(* IEC 61131-3 sources: study_plc/TimeStampFlat/content, 19 files *)

(* ---- main_prg.p~Variables~0000.var ---- *)
{ CustomGroupDefinition('a04e0da4-75a3-431c-a769-2ffcda83b779', '') }

VAR_EXTERNAL
    BUTTON_01 : BOOL { CustomGroupReference('a04e0da4-75a3-431c-a769-2ffcda83b779') } {Id('9d7c30a0-79f5-45dd-a2bb-9fe8afbc4b20')};
    LED : BOOL { CustomGroupReference('a04e0da4-75a3-431c-a769-2ffcda83b779') } {Id('db36f1cd-cd5f-4305-b62e-abae8295d826')};
END_VAR

VAR_GLOBAL
    bIsBlinking : BOOL { CustomGroupReference('a04e0da4-75a3-431c-a769-2ffcda83b779') } {Id('3276df67-48e3-40bd-b5cf-bc160ecd9fbf')};
    bLastButtonState : BOOL { CustomGroupReference('a04e0da4-75a3-431c-a769-2ffcda83b779') } {Id('10668f7e-212e-495e-babd-0d329f145ecd')};
    iBlinkCounter : INT { CustomGroupReference('a04e0da4-75a3-431c-a769-2ffcda83b779') } {Id('633e2c32-1f58-4700-8324-7b0311ee680d')};
    bCircleColor : BOOL { CustomGroupReference('a04e0da4-75a3-431c-a769-2ffcda83b779') } {Id('395212f8-a20c-46ba-a35b-0a9dcef59665')};
END_VAR

VAR_EXTERNAL
    counter : UINT { CustomGroupReference('a04e0da4-75a3-431c-a769-2ffcda83b779') } {Id('1701992e-3612-4291-8731-59990abaa8c7')};
    visual_counter : UINT { CustomGroupReference('a04e0da4-75a3-431c-a769-2ffcda83b779') } {Id('a891a596-3b4d-4571-8810-f9bcfd9d09ef')};
    tap_counter : UINT { CustomGroupReference('a04e0da4-75a3-431c-a769-2ffcda83b779') } {Id('a860a130-5121-4456-9e22-e20d3fb6a4d2')};
    TIMER : UINT { CustomGroupReference('a04e0da4-75a3-431c-a769-2ffcda83b779') } {Id('4b805dd1-1514-4363-b349-f760ae2ef950')};
    MESSAGE : BOOL { CustomGroupReference('a04e0da4-75a3-431c-a769-2ffcda83b779') } {Id('cdc6c82f-f8a2-467f-856e-2adb650c9a4f')};
    BUTTON_VIRTUAL : BOOL { CustomGroupReference('a04e0da4-75a3-431c-a769-2ffcda83b779') } {Id('e5aff69d-3d8e-4836-bed5-791e50e3ecc8')};
    buttonEdge : BOOL { CustomGroupReference('a04e0da4-75a3-431c-a769-2ffcda83b779') } {Id('871ce396-bc43-4252-ae3b-373c06ca63c2')};
    buttonCurrent : BOOL { CustomGroupReference('a04e0da4-75a3-431c-a769-2ffcda83b779') } {Id('1c2f3c40-a93c-4385-8462-9e9265ab8571')};
END_VAR

VAR
    FB21 : FB2 { CustomGroupReference('a04e0da4-75a3-431c-a769-2ffcda83b779') } {Id('54922560-dfac-4da8-a43d-80a38bc860ff')};
    FB22 : FB2 { CustomGroupReference('a04e0da4-75a3-431c-a769-2ffcda83b779') } {Id('0440c849-ac9a-4a62-b46c-6479d15f63f8')};
END_VAR

VAR_EXTERNAL
    TON_Blink : BOOL { CustomGroupReference('a04e0da4-75a3-431c-a769-2ffcda83b779') } {Id('319f1959-78a6-4cf2-81bc-d2dcea5df4e2')};
END_VAR

VAR
    FB23 : FB2 { CustomGroupReference('a04e0da4-75a3-431c-a769-2ffcda83b779') } {Id('546f7820-cb98-4ff5-a0ac-031b3fae9602')};
END_VAR

VAR_EXTERNAL
    blinkPeriod : UINT { CustomGroupReference('a04e0da4-75a3-431c-a769-2ffcda83b779') } {Id('be068b81-cd0d-40ca-b639-6780bc643a35')};
    TIME_TO_DINT : BOOL { CustomGroupReference('a04e0da4-75a3-431c-a769-2ffcda83b779') } {Id('cb415087-eb6f-4bb9-bdf8-b33e5cb765ee')};
    HMI_blinkPeriod : UINT { CustomGroupReference('a04e0da4-75a3-431c-a769-2ffcda83b779') } {Id('e62754f2-c4ad-4517-bcdd-83995e7e8a4c')};
END_VAR

VAR
    FB1 : FB { CustomGroupReference('a04e0da4-75a3-431c-a769-2ffcda83b779') } {Id('a21cc78b-fc91-401c-989f-5a3f00dbf2b6')};
    FB2 : FB { CustomGroupReference('a04e0da4-75a3-431c-a769-2ffcda83b779') } {Id('57562de0-dacc-42f6-93d3-63030d3f5b88')};
    FB3 : FB { CustomGroupReference('a04e0da4-75a3-431c-a769-2ffcda83b779') } {Id('74436edf-7137-4b89-ad20-294e1d8fb0ba')};
    FB4 : FB { CustomGroupReference('a04e0da4-75a3-431c-a769-2ffcda83b779') } {Id('58145396-09ad-45fc-99ee-1bc74df87d60')};
    FB5 : FB { CustomGroupReference('a04e0da4-75a3-431c-a769-2ffcda83b779') } {Id('605fd930-4c27-426e-82da-72f9c501b4c8')};
    UTC_in_Second1 : UTC_in_Second { CustomGroupReference('a04e0da4-75a3-431c-a769-2ffcda83b779') } {Id('561bc80b-119c-49be-b34c-1341fe2128dd')};
    UTC_in_Second2 : UTC_in_Second { CustomGroupReference('a04e0da4-75a3-431c-a769-2ffcda83b779') } {Id('187551ab-48a8-4595-8129-f3d7c5e3eedb')};
    UTC_in_Second3 : UTC_in_Second { CustomGroupReference('a04e0da4-75a3-431c-a769-2ffcda83b779') } {Id('8356627b-db3f-42a6-bade-665229c3f576')};
    UTC_in_Second4 : UTC_in_Second { CustomGroupReference('a04e0da4-75a3-431c-a769-2ffcda83b779') } {Id('4f025b1b-41c1-47cd-a402-58daae036f8e')};
    UTC_in_Second5 : UTC_in_Second { CustomGroupReference('a04e0da4-75a3-431c-a769-2ffcda83b779') } {Id('dae2764d-2f23-4bc9-8ce6-f3115f05c329')};
END_VAR

VAR_EXTERNAL
    TimestampMs : ULINT { CustomGroupReference('a04e0da4-75a3-431c-a769-2ffcda83b779') } {Id('bceea6ea-516d-42c0-a9bf-c36901277ad8')};
    ManualRTC : STRING { CustomGroupReference('a04e0da4-75a3-431c-a769-2ffcda83b779') } {Id('cec4a686-64db-40d8-a2d6-88bfda80289a')};
END_VAR

VAR
    UTC_in_Second6 : UTC_in_Second { CustomGroupReference('a04e0da4-75a3-431c-a769-2ffcda83b779') } {Id('34ce032f-88bf-46b0-9d48-2bfe1af360d8')};
END_VAR

(* ---- RES_3E844~GlobalVari~0000.var ---- *)
{ CustomGroupDefinition('fb84caa8-36a3-47d9-8bf0-95ff0e8a7b24', 'Default') }
{ CustomGroupDefinition('971398c9-e054-4349-a1d9-e00a1840c9f4', 'System Variables') }

VAR_GLOBAL
    BUTTON_01 : BOOL { CustomGroupReference('fb84caa8-36a3-47d9-8bf0-95ff0e8a7b24') } {Id('ff55c68f-4009-44e2-9111-0f6121b7f28e')};
    LED : BOOL { CustomGroupReference('fb84caa8-36a3-47d9-8bf0-95ff0e8a7b24') } {Id('a3518c0f-cfe9-4be8-920a-e2427bf7add7')};
    counter : UINT { CustomGroupReference('fb84caa8-36a3-47d9-8bf0-95ff0e8a7b24') } {Id('c758d767-5474-4789-9d22-781bfd7625a3')};
    bIsBlinking : BOOL { CustomGroupReference('fb84caa8-36a3-47d9-8bf0-95ff0e8a7b24') } {Id('41169e27-439a-46a2-bd00-94b8d785524f')};
    bLastButtonState : BOOL { CustomGroupReference('fb84caa8-36a3-47d9-8bf0-95ff0e8a7b24') } {Id('91fcfb61-3d5c-46c5-82ee-099172dd2d00')};
    visual_counter : UINT { CustomGroupReference('fb84caa8-36a3-47d9-8bf0-95ff0e8a7b24') } {Id('a5ecaf92-65ff-4985-a7f0-7e5144a773bc')};
    tap_counter : UINT { CustomGroupReference('fb84caa8-36a3-47d9-8bf0-95ff0e8a7b24') } {Id('7997c538-978c-452e-b505-3f3264cd3acb')};
    TIMER : UINT { CustomGroupReference('fb84caa8-36a3-47d9-8bf0-95ff0e8a7b24') } {Id('f51bd8e7-c0cd-421f-84a5-2d7e3e3f3667')};
    MESSAGE : BOOL { CustomGroupReference('fb84caa8-36a3-47d9-8bf0-95ff0e8a7b24') } {Id('3c2fc884-e19f-4beb-963f-04e6b1e4ad5f')};
    BUTTON_VIRTUAL : BOOL { CustomGroupReference('fb84caa8-36a3-47d9-8bf0-95ff0e8a7b24') } {Id('713492fe-22b0-4431-98a2-874f33c0214d')};
    buttonEdge : BOOL { CustomGroupReference('fb84caa8-36a3-47d9-8bf0-95ff0e8a7b24') } {Id('00cb1bf9-a75a-41ef-b864-ad11ab6e73bd')};
    buttonCurrent : BOOL { CustomGroupReference('fb84caa8-36a3-47d9-8bf0-95ff0e8a7b24') } {Id('a3914946-180c-4931-8b9b-c4945eb15232')};
END_VAR

VAR_CONFIG
    main_prg1.FB22.BUTTON_VIRTUAL : BOOL { InputLocation, CustomGroupReference('fb84caa8-36a3-47d9-8bf0-95ff0e8a7b24') } {Id('edaae17a-2832-4c67-ac45-b190593d386f')};
    main_prg1.FB21.BUTTON_VIRTUAL : BOOL { InputLocation, CustomGroupReference('fb84caa8-36a3-47d9-8bf0-95ff0e8a7b24') } {Id('30d0fe49-cb2f-4a7f-9de2-3afded5ed9e1')};
END_VAR

VAR_GLOBAL
    TIME_TO_DINT : BOOL { CustomGroupReference('fb84caa8-36a3-47d9-8bf0-95ff0e8a7b24') } {Id('c08fca2b-8685-447f-9b1d-964d4b9698af')};
    blinkPeriod : UINT { CustomGroupReference('fb84caa8-36a3-47d9-8bf0-95ff0e8a7b24') } {Id('a89eaa18-a4a3-4d70-906a-897dfc0313cd')};
    TON_Blink : BOOL { CustomGroupReference('fb84caa8-36a3-47d9-8bf0-95ff0e8a7b24') } {Id('687960f8-1ee0-416c-89ff-6b97b4efdd67')};
    HMI_blinkPeriod : UINT { CustomGroupReference('fb84caa8-36a3-47d9-8bf0-95ff0e8a7b24') } {Id('b5ffe9d3-7473-475f-903d-5c747d9fce23')};
    UINT_TO_TIME : BOOL { CustomGroupReference('fb84caa8-36a3-47d9-8bf0-95ff0e8a7b24') } {Id('56c9b7dd-8b0f-4834-bde7-82dd9a64a721')};
    PressStart : ULINT { CustomGroupReference('fb84caa8-36a3-47d9-8bf0-95ff0e8a7b24') } {Id('72598318-5edc-48d2-b4c1-9021699f7749')};
    PressTime : ULINT { CustomGroupReference('fb84caa8-36a3-47d9-8bf0-95ff0e8a7b24') } {Id('20e9929e-5bd7-41be-87ae-dc1696108355')};
    bButton : BOOL { CustomGroupReference('fb84caa8-36a3-47d9-8bf0-95ff0e8a7b24') } {Id('1b65edaf-19e7-4e96-9bb3-230a0c218b20')};
    BlinkReset : BOOL { CustomGroupReference('fb84caa8-36a3-47d9-8bf0-95ff0e8a7b24') } {Id('49695894-1423-4474-9eaa-ce1ad988c3f5')};
    test_us_1 : ULINT { CustomGroupReference('fb84caa8-36a3-47d9-8bf0-95ff0e8a7b24') } {Id('b3f01b14-7269-48aa-a0bd-12850281ca48')};
    test_us_2 : ULINT { CustomGroupReference('fb84caa8-36a3-47d9-8bf0-95ff0e8a7b24') } {Id('3fb0d77d-6462-4922-9943-9df0e6459224')};
    sTime : STRING { CustomGroupReference('fb84caa8-36a3-47d9-8bf0-95ff0e8a7b24') } {Id('b1cc24f8-6954-4e78-a01b-3fb7d85319ce')};
    bRTC_Ready : BOOL { CustomGroupReference('fb84caa8-36a3-47d9-8bf0-95ff0e8a7b24') } {Id('517801c9-9df0-49bf-9626-1117f62db573')};
    nLastBlink : ULINT { CustomGroupReference('fb84caa8-36a3-47d9-8bf0-95ff0e8a7b24') } {Id('f0fc7b48-9d55-4261-81d7-a2b4516753ed')};
    debug_toggle : INT { CustomGroupReference('fb84caa8-36a3-47d9-8bf0-95ff0e8a7b24') } {Id('4f1d6557-6d1f-4585-8eaa-0d52a0a13aa6')};
    bVirtualPulse : BOOL { CustomGroupReference('fb84caa8-36a3-47d9-8bf0-95ff0e8a7b24') } {Id('1a3d1420-8400-4ed1-ae9a-b1be359f92a0')};
    bLastVirtual : BOOL { CustomGroupReference('fb84caa8-36a3-47d9-8bf0-95ff0e8a7b24') } {Id('2a59c38b-860d-41cc-b434-8815cd6eb838')};
    bVirtTrig : BOOL { CustomGroupReference('fb84caa8-36a3-47d9-8bf0-95ff0e8a7b24') } {Id('2d522a4e-02e2-4d08-8e87-e2abe91557be')};
    bLastButton : BOOL { CustomGroupReference('fb84caa8-36a3-47d9-8bf0-95ff0e8a7b24') } {Id('e926f615-f63b-44f9-a00b-60eff743de3b')};
    rTrigVirt : BOOL { CustomGroupReference('fb84caa8-36a3-47d9-8bf0-95ff0e8a7b24') } {Id('95be6528-0073-416e-87ec-9c3c74cfbb9f')};
    rTrigPhys : BOOL { CustomGroupReference('fb84caa8-36a3-47d9-8bf0-95ff0e8a7b24') } {Id('f3b9ac2f-ae6f-4cfb-9b98-34b4fd9e6e43')};
    bWaitForRelease : BOOL { CustomGroupReference('fb84caa8-36a3-47d9-8bf0-95ff0e8a7b24') } {Id('cee13b13-a0ba-47f2-85b5-a1153d2bfc4d')};
    bLastPhys : BOOL { CustomGroupReference('fb84caa8-36a3-47d9-8bf0-95ff0e8a7b24') } {Id('2c93ea6f-76fc-46c1-8245-239521de7509')};
    bLastVirt : BOOL { CustomGroupReference('fb84caa8-36a3-47d9-8bf0-95ff0e8a7b24') } {Id('e15edbd4-dc20-4abf-a76b-535e03ed0216')};
    bVirtOneShot : BOOL { CustomGroupReference('fb84caa8-36a3-47d9-8bf0-95ff0e8a7b24') } {Id('180e95ba-7660-42f3-ab82-8aa1f4af8f65')};
    bPhysOneShot : BOOL { CustomGroupReference('fb84caa8-36a3-47d9-8bf0-95ff0e8a7b24') } {Id('b17a499a-a16a-4e07-a451-effc40a9126b')};
    bAnyPress : BOOL { CustomGroupReference('fb84caa8-36a3-47d9-8bf0-95ff0e8a7b24') } {Id('0312dcf0-9424-407f-a37e-e022e10eb398')};
    bVirtOld : BOOL { CustomGroupReference('fb84caa8-36a3-47d9-8bf0-95ff0e8a7b24') } {Id('ca6bffc0-4800-4d66-aefe-acab4512e9e1')};
    TRIM : BOOL { CustomGroupReference('fb84caa8-36a3-47d9-8bf0-95ff0e8a7b24') } {Id('6c8b045d-0aab-487b-b1ad-cb855cf61a63')};
    bRTCReady : BOOL { CustomGroupReference('fb84caa8-36a3-47d9-8bf0-95ff0e8a7b24') } {Id('cb59c76f-3031-4077-8f90-714e8f7a8c8b')};
    TimestampMs : ULINT { CustomGroupReference('fb84caa8-36a3-47d9-8bf0-95ff0e8a7b24') } {Id('84cfde2f-c5c3-4348-808e-c1645fed4d81')};
    TimeZone : INT { CustomGroupReference('fb84caa8-36a3-47d9-8bf0-95ff0e8a7b24') } {Id('1288d1f3-3ab3-4651-8a72-0030e0acb8f2')};
    nTimeZoneOffset : INT { CustomGroupReference('fb84caa8-36a3-47d9-8bf0-95ff0e8a7b24') } {Id('d52ba4d7-7e69-49ff-be6d-e2df38c82290')};
    sOutputDate : STRING { CustomGroupReference('fb84caa8-36a3-47d9-8bf0-95ff0e8a7b24') } {Id('045fa39e-965c-40ad-9d1c-b2ae0bfc88d7')};
    ulInputMS : ULINT { CustomGroupReference('fb84caa8-36a3-47d9-8bf0-95ff0e8a7b24') } {Id('57f31c1f-ce8e-4e9a-a54f-91a1926557d9')};
    sCustomDate : STRING { CustomGroupReference('fb84caa8-36a3-47d9-8bf0-95ff0e8a7b24') } {Id('7e064ee7-e4f6-4547-b34e-d6702123f182')};
END_VAR

VAR_CONFIG
    main_prg1.UTC_in_Second5.DaysInMonth : INT { InputLocation, CustomGroupReference('fb84caa8-36a3-47d9-8bf0-95ff0e8a7b24') } {Id('0b54d02d-88a7-4f64-a714-37ba5a4d2863')};
    main_prg1.UTC_in_Second4.DaysInMonth : INT { InputLocation, CustomGroupReference('fb84caa8-36a3-47d9-8bf0-95ff0e8a7b24') } {Id('c5c31dc5-7259-4959-b722-8cf1dc1f7ee6')};
    main_prg1.UTC_in_Second3.DaysInMonth : INT { InputLocation, CustomGroupReference('fb84caa8-36a3-47d9-8bf0-95ff0e8a7b24') } {Id('babf101c-e82f-4d04-9ab9-a52ee78929ee')};
    main_prg1.UTC_in_Second2.DaysInMonth : INT { InputLocation, CustomGroupReference('fb84caa8-36a3-47d9-8bf0-95ff0e8a7b24') } {Id('af5cefd6-4978-424f-95ca-eec832feb9ce')};
    main_prg1.UTC_in_Second1.DaysInMonth : INT { InputLocation, CustomGroupReference('fb84caa8-36a3-47d9-8bf0-95ff0e8a7b24') } {Id('cc2d7a49-7d34-4f98-8bad-cdc305743582')};
END_VAR

VAR_GLOBAL
    sTmp : BOOL { CustomGroupReference('fb84caa8-36a3-47d9-8bf0-95ff0e8a7b24') } {Id('52421147-2409-4498-864b-2a037dc35c02')};
    sTmp2 : BOOL { CustomGroupReference('fb84caa8-36a3-47d9-8bf0-95ff0e8a7b24') } {Id('9060f604-83ec-4e2e-8322-d678c276741c')};
    sYy : STRING { CustomGroupReference('fb84caa8-36a3-47d9-8bf0-95ff0e8a7b24') } {Id('4c9b6b92-2451-4146-be8f-061a9e49ac85')};
    sMo : STRING { CustomGroupReference('fb84caa8-36a3-47d9-8bf0-95ff0e8a7b24') } {Id('2338197b-f5fd-40a7-9e1a-48057039073d')};
    nMonthDays : INT { CustomGroupReference('fb84caa8-36a3-47d9-8bf0-95ff0e8a7b24') } {Id('afdd7226-203a-4163-8ab4-f50e96edd491')};
    UseManualRTC : BOOL { CustomGroupReference('fb84caa8-36a3-47d9-8bf0-95ff0e8a7b24') } {Id('b1822fe9-4cea-4d3a-b67e-cfc11819dcf7')};
    ManualRTC : STRING { CustomGroupReference('fb84caa8-36a3-47d9-8bf0-95ff0e8a7b24') } {Id('03a235b0-b550-43e6-9f6e-0f7724ebddc2')};
    TimezoneOffset : INT { CustomGroupReference('fb84caa8-36a3-47d9-8bf0-95ff0e8a7b24') } {Id('24b06e47-b007-45e8-8735-7f3f73c4efa8')};
END_VAR

VAR_CONFIG
    main_prg1.UTC_in_Second6.DaysInMonth : INT { InputLocation, CustomGroupReference('fb84caa8-36a3-47d9-8bf0-95ff0e8a7b24') } {Id('18a8efd7-5980-422a-b2ec-fcc23db0160e')};
END_VAR

VAR_GLOBAL
    PND_S1_PLC_RUN : BOOL { SystemVariable, CustomGroupReference('971398c9-e054-4349-a1d9-e00a1840c9f4') } {Id('a8109aaa-718e-4ad7-9ef6-414f49af5f2c')}; (*Higher level PLC in RUN*)
    PND_S1_VALID_DATA_CYCLE : BOOL { SystemVariable, CustomGroupReference('971398c9-e054-4349-a1d9-e00a1840c9f4') } {Id('e4636e3b-85f5-4518-8ba6-e632d844bd79')}; (*Connection to Profinet-Controller*)
    PND_S1_OUTPUT_STATUS_GOOD : BOOL { SystemVariable, CustomGroupReference('971398c9-e054-4349-a1d9-e00a1840c9f4') } {Id('9e967e71-8e8f-40d9-aae6-a7f87e15c1dc')}; (*IOP status of the higher-level control system*)
    PND_S1_INPUT_STATUS_GOOD : BOOL { SystemVariable, CustomGroupReference('971398c9-e054-4349-a1d9-e00a1840c9f4') } {Id('b1e203c1-a3c2-41a1-8f15-cba8c60dc0f2')}; (*IOC status of the higher-level control system*)
    PND_S1_DATA_LENGTH : WORD { SystemVariable, CustomGroupReference('971398c9-e054-4349-a1d9-e00a1840c9f4') } {Id('c69796fa-e3a1-44c3-8dc7-85a985bef384')}; (*Process data length*)
    PND_S1_OUTPUTS : PND_IO_512 { SystemVariable, CustomGroupReference('971398c9-e054-4349-a1d9-e00a1840c9f4'), Assignable(IsWritable := True), Origin('epd056') } {Id('871d0d2f-9f74-43af-844e-7e8a0b6267c3')}; (*Output process data*)
    PND_S1_INPUTS : PND_IO_512 { SystemVariable, CustomGroupReference('971398c9-e054-4349-a1d9-e00a1840c9f4') } {Id('26de38c2-6476-4746-acc5-bee0b9f2dbfa')}; (*Input process data*)
    PND_IO_DRIVEN_BY_PLC : INT { SystemVariable, CustomGroupReference('971398c9-e054-4349-a1d9-e00a1840c9f4') } {Id('00739d06-8933-4fec-8048-b3cebcbc2058')};
    AXIO_DIAG_STATUS_REG_HI : BYTE { SystemVariable, CustomGroupReference('971398c9-e054-4349-a1d9-e00a1840c9f4') } {Id('4f9c59a1-643a-4475-a439-ad1cf8561ad6')};
    AXIO_DIAG_STATUS_REG_LOW : BYTE { SystemVariable, CustomGroupReference('971398c9-e054-4349-a1d9-e00a1840c9f4') } {Id('eae2279f-0f04-4890-a0bf-b55fad2d0afa')};
    AXIO_DIAG_PARAM_REG_HI : BYTE { SystemVariable, CustomGroupReference('971398c9-e054-4349-a1d9-e00a1840c9f4') } {Id('0caba1d5-e173-4e1b-b805-00d054efa100')};
    AXIO_DIAG_PARAM_REG_LOW : BYTE { SystemVariable, CustomGroupReference('971398c9-e054-4349-a1d9-e00a1840c9f4') } {Id('67315ed2-b4f9-44bb-859d-233dd4b3c9bb')};
    AXIO_DIAG_PARAM_2_REG_HI : BYTE { SystemVariable, CustomGroupReference('971398c9-e054-4349-a1d9-e00a1840c9f4') } {Id('981f8143-c142-4f6c-ae92-2b18592edb2f')};
    AXIO_DIAG_PARAM_2_REG_LOW : BYTE { SystemVariable, CustomGroupReference('971398c9-e054-4349-a1d9-e00a1840c9f4') } {Id('f7a3077a-9e70-458b-acdb-2714bd9d86a3')};
    AXIO_DIAG_STATUS_REG_PF : BOOL { SystemVariable, CustomGroupReference('971398c9-e054-4349-a1d9-e00a1840c9f4') } {Id('c49d1a45-1fcc-4ae2-b55e-619e93c6f775')};
    AXIO_DIAG_STATUS_REG_BUS : BOOL { SystemVariable, CustomGroupReference('971398c9-e054-4349-a1d9-e00a1840c9f4') } {Id('17b3305e-f37e-4a9d-94a4-5a3d9ca6ad1a')};
    AXIO_DIAG_STATUS_REG_RUN : BOOL { SystemVariable, CustomGroupReference('971398c9-e054-4349-a1d9-e00a1840c9f4') } {Id('79b3d4f7-46d4-4c7b-aa70-24e501b5afeb')};
    AXIO_DIAG_STATUS_REG_ACT : BOOL { SystemVariable, CustomGroupReference('971398c9-e054-4349-a1d9-e00a1840c9f4') } {Id('a0315e8d-4040-4508-b50d-7fa5ad74f7a1')};
    AXIO_DIAG_STATUS_REG_RDY : BOOL { SystemVariable, CustomGroupReference('971398c9-e054-4349-a1d9-e00a1840c9f4') } {Id('c8b37275-37bf-40c1-94c8-2d91ca269131')};
    AXIO_DIAG_STATUS_REG_SYSFAIL : BOOL { SystemVariable, CustomGroupReference('971398c9-e054-4349-a1d9-e00a1840c9f4') } {Id('a230509c-5098-49c0-94c0-ee773a64e2de')};
    AXIO_DIAG_STATUS_REG_PW : BOOL { SystemVariable, CustomGroupReference('971398c9-e054-4349-a1d9-e00a1840c9f4') } {Id('67e3682d-83f4-44e0-ac88-2f95bae65960')};
    IB_DIAG_STATUS_REG_HI : BYTE { SystemVariable, CustomGroupReference('971398c9-e054-4349-a1d9-e00a1840c9f4'), Assignable(IsWritable := True), Origin('epdib1') } {Id('870f34b1-cbfb-4a12-9a3a-674532964b8e')};
    IB_DIAG_STATUS_REG_LOW : BYTE { SystemVariable, CustomGroupReference('971398c9-e054-4349-a1d9-e00a1840c9f4'), Assignable(IsWritable := True), Origin('epdib2') } {Id('6aca7f7b-4495-47d2-b6c9-b992b56c11ef')};
    IB_DIAG_STATUS_REG_SYSFAIL : BOOL { SystemVariable, CustomGroupReference('971398c9-e054-4349-a1d9-e00a1840c9f4'), Assignable(IsWritable := True), Origin('epdib3') } {Id('8836a82b-e65b-4bcd-bdda-0e80ed208fef')};
    IB_DIAG_STATUS_REG_WARN : BOOL { SystemVariable, CustomGroupReference('971398c9-e054-4349-a1d9-e00a1840c9f4'), Assignable(IsWritable := True), Origin('epdib4') } {Id('590ff5fc-a4de-4153-abff-4c319033e938')};
    IB_DIAG_STATUS_REG_QUAL : BOOL { SystemVariable, CustomGroupReference('971398c9-e054-4349-a1d9-e00a1840c9f4'), Assignable(IsWritable := True), Origin('epdib5') } {Id('016a54f4-214c-4108-9e23-713c4e30776f')};
    IB_DIAG_STATUS_REG_USER : BOOL { SystemVariable, CustomGroupReference('971398c9-e054-4349-a1d9-e00a1840c9f4'), Assignable(IsWritable := True), Origin('epdib6') } {Id('436892d9-24f4-4bde-b365-39ce805afbcb')};
    IB_DIAG_STATUS_REG_PF : BOOL { SystemVariable, CustomGroupReference('971398c9-e054-4349-a1d9-e00a1840c9f4'), Assignable(IsWritable := True), Origin('epdib7') } {Id('9db6ace2-a1c0-4f18-b2cc-23c676225b79')};
    IB_DIAG_STATUS_REG_BUS : BOOL { SystemVariable, CustomGroupReference('971398c9-e054-4349-a1d9-e00a1840c9f4'), Assignable(IsWritable := True), Origin('epdib8') } {Id('69b61899-e7d4-45a0-a00c-0858c7e6436a')};
    IB_DIAG_STATUS_REG_CTRL : BOOL { SystemVariable, CustomGroupReference('971398c9-e054-4349-a1d9-e00a1840c9f4'), Assignable(IsWritable := True), Origin('epdib9') } {Id('ea44b33b-9512-4145-9c83-f5fc837d58a5')};
    IB_DIAG_STATUS_REG_DTC : BOOL { SystemVariable, CustomGroupReference('971398c9-e054-4349-a1d9-e00a1840c9f4'), Assignable(IsWritable := True), Origin('epdib10') } {Id('56dd80ec-9280-441e-bd4f-2ac40a37e096')};
    IB_DIAG_STATUS_REG_RUN : BOOL { SystemVariable, CustomGroupReference('971398c9-e054-4349-a1d9-e00a1840c9f4'), Assignable(IsWritable := True), Origin('epdib11') } {Id('c59a357f-adc9-49ca-a807-b1c10b0d67a2')};
    IB_DIAG_STATUS_REG_ACT : BOOL { SystemVariable, CustomGroupReference('971398c9-e054-4349-a1d9-e00a1840c9f4'), Assignable(IsWritable := True), Origin('epdib12') } {Id('e3ecf724-72f2-4fe3-be90-c451638ac496')};
    IB_DIAG_STATUS_REG_RDY : BOOL { SystemVariable, CustomGroupReference('971398c9-e054-4349-a1d9-e00a1840c9f4'), Assignable(IsWritable := True), Origin('epdib13') } {Id('5c061d11-60fc-4a47-a192-85e8775eb15f')};
    IB_DIAG_PARAM_REG_HI : BYTE { SystemVariable, CustomGroupReference('971398c9-e054-4349-a1d9-e00a1840c9f4'), Assignable(IsWritable := True), Origin('epdib14') } {Id('38a23e35-1cd8-4d9c-96d6-810c618d5526')};
    IB_DIAG_PARAM_REG_LOW : BYTE { SystemVariable, CustomGroupReference('971398c9-e054-4349-a1d9-e00a1840c9f4'), Assignable(IsWritable := True), Origin('epdib15') } {Id('5b495f5b-d26e-4cff-836b-0fe238b1654d')};
    IB_DIAG_PARAM_2_REG_HI : BYTE { SystemVariable, CustomGroupReference('971398c9-e054-4349-a1d9-e00a1840c9f4'), Assignable(IsWritable := True), Origin('epdib16') } {Id('317a6edf-8d30-4505-8601-eb0d20c3c6e2')};
    IB_DIAG_PARAM_2_REG_LOW : BYTE { SystemVariable, CustomGroupReference('971398c9-e054-4349-a1d9-e00a1840c9f4'), Assignable(IsWritable := True), Origin('epdib17') } {Id('83c1a718-f3e7-4cc0-841f-c1e2233f8d2e')};
    ESM_DATA : ESM_DAT { SystemVariable, CustomGroupReference('971398c9-e054-4349-a1d9-e00a1840c9f4'), Assignable(IsWritable := True), Origin('epd100') } {Id('74de6c32-cd1d-4959-95c5-ec365806a030')};
    RTC : RTC_TYPE { SystemVariable, CustomGroupReference('971398c9-e054-4349-a1d9-e00a1840c9f4') } {Id('3c52e428-0cdb-4c6c-bc54-e6da1e8c50fe')};
    DEVICE_STATE : DEVICE_STATE_2152_TYPE { SystemVariable, CustomGroupReference('971398c9-e054-4349-a1d9-e00a1840c9f4') } {Id('1129891b-b5a9-4d3b-b9a0-4936e33ad606')};
    USER_PARTITION : PARTITION_INFO { SystemVariable, CustomGroupReference('971398c9-e054-4349-a1d9-e00a1840c9f4') } {Id('4b7f6b3b-3696-419a-a21a-ce7cb6ceb9db')};
    PNIO_SYSTEM_BF : BOOL { SystemVariable, CustomGroupReference('971398c9-e054-4349-a1d9-e00a1840c9f4') } {Id('ea9f164c-d192-4b60-b66f-cf87b53d5e5b')};
    PNIO_SYSTEM_SF : BOOL { SystemVariable, CustomGroupReference('971398c9-e054-4349-a1d9-e00a1840c9f4') } {Id('de2bebd9-d808-496f-954f-38ec8ace12e8')};
    PNIO_MAINTENANCE_DEMANDED : BOOL { SystemVariable, CustomGroupReference('971398c9-e054-4349-a1d9-e00a1840c9f4') } {Id('4c4c4e79-3946-4f32-b468-22905a5c8f5f')};
    PNIO_MAINTENANCE_REQUIRED : BOOL { SystemVariable, CustomGroupReference('971398c9-e054-4349-a1d9-e00a1840c9f4') } {Id('0dfc99eb-ecfe-45c6-afb8-64b2d7705677')};
    PNIO_CONFIG_STATUS : WORD { SystemVariable, CustomGroupReference('971398c9-e054-4349-a1d9-e00a1840c9f4') } {Id('c34f805f-b5c2-44af-bb0f-7c49d4666c2f')};
    PNIO_CONFIG_STATUS_ACTIVE : BOOL { SystemVariable, CustomGroupReference('971398c9-e054-4349-a1d9-e00a1840c9f4') } {Id('d08caa2c-5061-4764-8b36-3a6b79934353')};
    PNIO_CONFIG_STATUS_READY : BOOL { SystemVariable, CustomGroupReference('971398c9-e054-4349-a1d9-e00a1840c9f4') } {Id('25aaf986-14d2-455e-8fb6-e8e35bd65063')};
    PNIO_CONFIG_STATUS_CFG_FAULT : BOOL { SystemVariable, CustomGroupReference('971398c9-e054-4349-a1d9-e00a1840c9f4') } {Id('7223f36b-f452-48c9-a964-10165bc7f0a7')};
    PNIO_FORCE_FAILSAFE : BOOL { SystemVariable, CustomGroupReference('971398c9-e054-4349-a1d9-e00a1840c9f4'), Assignable(IsWritable := True), Origin('epd145') } {Id('e1337b3e-a988-48a5-87ec-e8461474d15f')};
    PNIO_FORCE_PRIMARY : BOOL { SystemVariable, CustomGroupReference('971398c9-e054-4349-a1d9-e00a1840c9f4'), Assignable(IsWritable := True), Origin('epd159') } {Id('2e5ecda8-89ea-46e5-93c1-a46de4cc3fa2')};
    IP_ACTIVE_SOCKETS AT %MW1.30000 : UINT { SystemVariable, CustomGroupReference('971398c9-e054-4349-a1d9-e00a1840c9f4') } {Id('f10f644a-6de6-4578-8707-c22090109bfe')};
    TLS_ACTIVE_SOCKETS AT %MW1.30100 : UINT { SystemVariable, CustomGroupReference('971398c9-e054-4349-a1d9-e00a1840c9f4') } {Id('b614145a-4322-4555-8406-73f21140d7b8')};
    HMI_STATUS2 : HMI_STATUS_TYPE2 { SystemVariable, CustomGroupReference('971398c9-e054-4349-a1d9-e00a1840c9f4') } {Id('a142712d-5d2f-43da-8c93-deb2c52e6525')};
    HMI_CONTROL : HMI_CONTROL_TYPE { SystemVariable, CustomGroupReference('971398c9-e054-4349-a1d9-e00a1840c9f4'), Assignable(IsWritable := True), Origin('epd151') } {Id('9e0c5809-738c-47e0-98c3-088c020b755a')};
    EIPD_INPUTS : EIPD_IO_ARRAY { SystemVariable, CustomGroupReference('971398c9-e054-4349-a1d9-e00a1840c9f4') } {Id('876bd6bd-0ab9-42a0-8c1a-986f5c03e455')};
    EIPD_OUTPUTS : EIPD_IO_ARRAY { SystemVariable, CustomGroupReference('971398c9-e054-4349-a1d9-e00a1840c9f4'), Assignable(IsWritable := True), Origin('epd153') } {Id('ee7a2a99-783e-472f-9cae-c449c38f3da8')};
    EIPD_VALID_DATA_CYCLE : BOOL { SystemVariable, CustomGroupReference('971398c9-e054-4349-a1d9-e00a1840c9f4') } {Id('7ef7e2c3-a29c-4fb9-b6b9-6d2708115b6c')};
    EIPD_PEER_IDLE : BOOL { SystemVariable, CustomGroupReference('971398c9-e054-4349-a1d9-e00a1840c9f4') } {Id('ece7b39f-4744-4856-ab49-ac0106b18a4c')};
    EIPD_PEER_RUN : BOOL { SystemVariable, CustomGroupReference('971398c9-e054-4349-a1d9-e00a1840c9f4') } {Id('9a9a04d6-b3b6-4f81-8713-309c56ef942d')};
    EIPD_OUTPUTS_LENGTH : WORD { SystemVariable, CustomGroupReference('971398c9-e054-4349-a1d9-e00a1840c9f4') } {Id('852a06b4-24e7-4a6a-a226-9832b61a169c')};
    EIPD_INPUTS_LENGTH : WORD { SystemVariable, CustomGroupReference('971398c9-e054-4349-a1d9-e00a1840c9f4') } {Id('2475dd19-5aff-47a6-ba79-1133d75b5c3e')};
    PLC_CRC_PRJ AT %ML1.10000 : ULINT { SystemVariable, CustomGroupReference('971398c9-e054-4349-a1d9-e00a1840c9f4') } {Id('41b139bc-2750-4dde-b5bf-ab57e61bf63e')};
END_VAR

(* ---- FB.pou~Code~0000.st ---- *)
// время с контроллера
fbRTC(EN := TRUE, CDT => sTime, Q => bRTC_Ready);

// парс
fbParseTime(
    sTime := sTime,
    Year => nYear,
    Month => nMonth,
    Day => nDay,
    Hour => nHour,
    Minute => nMinute,
    Second => nSecond,
    Millisecond => nMS,
    Valid => bTimeValid
);

// количество дней от 1970
nDays := 0;

FOR i := 1970 TO nYear - 1 DO
    IF ((i MOD 4 = 0) AND (i MOD 100 <> 0)) OR (i MOD 400 = 0) THEN
        nDays := nDays + 366;
    ELSE
        nDays := nDays + 365;
    END_IF;
END_FOR;

// добавляем дни за полные месяцы
IF nMonth > 1 THEN nDays := nDays + 31; END_IF;
IF nMonth > 2 THEN
    IF ((nYear MOD 4 = 0) AND (nYear MOD 100 <> 0)) OR (nYear MOD 400 = 0) THEN
        nDays := nDays + 29;
    ELSE
        nDays := nDays + 28;
    END_IF;
END_IF;
IF nMonth > 3 THEN nDays := nDays + 31; END_IF;
IF nMonth > 4 THEN nDays := nDays + 30; END_IF;
IF nMonth > 5 THEN nDays := nDays + 31; END_IF;
IF nMonth > 6 THEN nDays := nDays + 30; END_IF;
IF nMonth > 7 THEN nDays := nDays + 31; END_IF;
IF nMonth > 8 THEN nDays := nDays + 31; END_IF;
IF nMonth > 9 THEN nDays := nDays + 30; END_IF;
IF nMonth > 10 THEN nDays := nDays + 31; END_IF;
IF nMonth > 11 THEN nDays := nDays + 30; END_IF;

// добавим дни текущего месяца
nDays := nDays + (nDay - 1);

// перевод всё в мс
TimestampMs :=
    DINT_TO_ULINT(nDays) * 86400000 +
    INT_TO_ULINT(nHour) * 3600000 +
    INT_TO_ULINT(nMinute) * 60000 +
    INT_TO_ULINT(nSecond) * 1000 +
    INT_TO_ULINT(nMS);

// сброс
IF BlinkReset THEN
    bIsBlinking := FALSE;
    visual_counter := 0;
    tap_counter := 0;
    LED := FALSE;
    nLastBlink := 0;
    bWaitForRelease := FALSE;
    BlinkReset := FALSE;
END_IF

(* ---- FB.pou~Variables~0000.var ---- *)
{ CustomGroupDefinition('d879d638-e7f1-4a28-a2ab-b4cf2ec7bb4a', '') }

VAR_INPUT
    BUTTON_01 : BOOL { CustomGroupReference('d879d638-e7f1-4a28-a2ab-b4cf2ec7bb4a') } {Id('4e0719f1-9a21-49b0-ab1a-7bca753de8bf')};
    BUTTON_VIRTUAL : BOOL { CustomGroupReference('d879d638-e7f1-4a28-a2ab-b4cf2ec7bb4a') } {Id('16b13fcd-91ca-4fbd-bce8-5329faf97148')};
END_VAR

VAR_OUTPUT
    LED : BOOL { CustomGroupReference('d879d638-e7f1-4a28-a2ab-b4cf2ec7bb4a') } {Id('35a522c3-a831-4de5-82d7-ae5b3c0dd537')};
    MESSAGE : BOOL { CustomGroupReference('d879d638-e7f1-4a28-a2ab-b4cf2ec7bb4a') } {Id('fb214dee-66f6-463f-9713-862a6108447e')};
END_VAR

VAR
    PressStart : ULINT { CustomGroupReference('d879d638-e7f1-4a28-a2ab-b4cf2ec7bb4a') } {Id('ae5033d3-fed2-43d0-adf6-ccfa772e577f')};
    PressTime : ULINT { CustomGroupReference('d879d638-e7f1-4a28-a2ab-b4cf2ec7bb4a') } {Id('67c05195-0624-4f5b-a4a4-63254ac533c9')};
    bButton : BOOL { CustomGroupReference('d879d638-e7f1-4a28-a2ab-b4cf2ec7bb4a') } {Id('a6f25af8-da50-4153-a6f2-77781ed29851')};
    bLastButtonState : BOOL { CustomGroupReference('d879d638-e7f1-4a28-a2ab-b4cf2ec7bb4a') } {Id('4f0463dc-8f77-4d98-87a2-aa94574099e2')};
    bIsBlinking : BOOL { CustomGroupReference('d879d638-e7f1-4a28-a2ab-b4cf2ec7bb4a') } {Id('b9bf86c3-b159-4991-9861-6f5314b0321c')};
    BlinkReset : BOOL { CustomGroupReference('d879d638-e7f1-4a28-a2ab-b4cf2ec7bb4a') } {Id('7e2c85d6-cf72-46e0-b9a5-424ab27580a5')};
    TON_Blink : TON { CustomGroupReference('d879d638-e7f1-4a28-a2ab-b4cf2ec7bb4a') } {Id('197c8782-f631-4ffa-a13c-2cd90675b891')};
END_VAR

VAR_EXTERNAL
    visual_counter : UINT { CustomGroupReference('d879d638-e7f1-4a28-a2ab-b4cf2ec7bb4a') } {Id('ed5c4f7a-75fb-4186-8b26-909a554518ed')};
    tap_counter : UINT { CustomGroupReference('d879d638-e7f1-4a28-a2ab-b4cf2ec7bb4a') } {Id('8e4fb33c-aed4-48aa-8ee2-6ffca498c8a3')};
END_VAR

VAR
    dummy : ULINT { CustomGroupReference('d879d638-e7f1-4a28-a2ab-b4cf2ec7bb4a') } {Id('206ff9a5-ceb4-427d-bf17-5ced64b3d33f')};
    fbRTC : RTC_S { CustomGroupReference('d879d638-e7f1-4a28-a2ab-b4cf2ec7bb4a') } {Id('689cfebd-229e-4b45-8dd0-65fa994717f3')};
END_VAR

VAR_EXTERNAL
    sTime : STRING { CustomGroupReference('d879d638-e7f1-4a28-a2ab-b4cf2ec7bb4a') } {Id('91bb18d7-44e6-4613-a079-9ddb7a779d7d')};
    bRTC_Ready : BOOL { CustomGroupReference('d879d638-e7f1-4a28-a2ab-b4cf2ec7bb4a') } {Id('c414b8d8-2513-4024-ae96-ac7c04fab89d')};
    nLastBlink : ULINT { CustomGroupReference('d879d638-e7f1-4a28-a2ab-b4cf2ec7bb4a') } {Id('cb3e5d71-9c5a-4d71-8037-b20658097fc0')};
    debug_toggle : INT { CustomGroupReference('d879d638-e7f1-4a28-a2ab-b4cf2ec7bb4a') } {Id('2072d667-54cb-490a-b42a-0cae67e0ad60')};
    bVirtualPulse : BOOL { CustomGroupReference('d879d638-e7f1-4a28-a2ab-b4cf2ec7bb4a') } {Id('6798c4c2-251a-4f23-8819-dd3632552722')};
    bLastVirtual : BOOL { CustomGroupReference('d879d638-e7f1-4a28-a2ab-b4cf2ec7bb4a') } {Id('53ac58ec-322e-422e-aaf0-86794f043220')};
    bVirtTrig : BOOL { CustomGroupReference('d879d638-e7f1-4a28-a2ab-b4cf2ec7bb4a') } {Id('57ff68d4-c262-4da7-a951-55c5bc88e074')};
    bLastButton : BOOL { CustomGroupReference('d879d638-e7f1-4a28-a2ab-b4cf2ec7bb4a') } {Id('3a263dd4-d980-4a3f-9643-d60d3c28d595')};
END_VAR

VAR
    rTrigVirt : R_TRIG { CustomGroupReference('d879d638-e7f1-4a28-a2ab-b4cf2ec7bb4a') } {Id('c425a54f-4ffb-481e-90de-1a6ced1796a6')};
    rTrigPhys : R_TRIG { CustomGroupReference('d879d638-e7f1-4a28-a2ab-b4cf2ec7bb4a') } {Id('19454729-86e8-4c30-9d95-3b307f57250b')};
END_VAR

VAR_EXTERNAL
    bWaitForRelease : BOOL { CustomGroupReference('d879d638-e7f1-4a28-a2ab-b4cf2ec7bb4a') } {Id('f76a665a-d697-43fa-a6b8-18f2ea8978be')};
    bLastPhys : BOOL { CustomGroupReference('d879d638-e7f1-4a28-a2ab-b4cf2ec7bb4a') } {Id('531aa2b4-5bc9-4d3d-a0a4-8ab213c87f93')};
    bLastVirt : BOOL { CustomGroupReference('d879d638-e7f1-4a28-a2ab-b4cf2ec7bb4a') } {Id('922be82b-f033-4ced-a705-cc1dc33cad68')};
    bVirtOneShot : BOOL { CustomGroupReference('d879d638-e7f1-4a28-a2ab-b4cf2ec7bb4a') } {Id('f4a75110-e32c-4b99-910e-0a3c7e07d5e2')};
    bPhysOneShot : BOOL { CustomGroupReference('d879d638-e7f1-4a28-a2ab-b4cf2ec7bb4a') } {Id('2b008f14-1972-47cd-b851-4c2584ccefca')};
    bAnyPress : BOOL { CustomGroupReference('d879d638-e7f1-4a28-a2ab-b4cf2ec7bb4a') } {Id('3e3f621f-cc8c-478e-9c93-b44046d7376d')};
    bVirtOld : BOOL { CustomGroupReference('d879d638-e7f1-4a28-a2ab-b4cf2ec7bb4a') } {Id('68ce2f51-fafa-4cf1-844d-ab73b71ba07b')};
    blinkPeriod : UINT { CustomGroupReference('d879d638-e7f1-4a28-a2ab-b4cf2ec7bb4a') } {Id('a56961bd-2c08-4691-832b-77807cfcc86c')};
END_VAR

VAR
    fbParseTime : ParseRTC_Time { CustomGroupReference('d879d638-e7f1-4a28-a2ab-b4cf2ec7bb4a') } {Id('cce46eaa-d2db-4059-a9d3-e31aabe5a6af')};
    nYear : INT { CustomGroupReference('d879d638-e7f1-4a28-a2ab-b4cf2ec7bb4a') } {Id('777e47e4-9352-417e-9871-07007a5dc2b9')};
    nMonth : INT { CustomGroupReference('d879d638-e7f1-4a28-a2ab-b4cf2ec7bb4a') } {Id('17b63c43-e232-4cd0-9329-bc6ecde28367')};
    nDay : INT { CustomGroupReference('d879d638-e7f1-4a28-a2ab-b4cf2ec7bb4a') } {Id('610470b4-db4d-4a77-8adb-1317351dabfa')};
    nMinute : INT { CustomGroupReference('d879d638-e7f1-4a28-a2ab-b4cf2ec7bb4a') } {Id('3cfe0860-a69c-4d2b-9aed-adbf35338e72')};
    nSecond : INT { CustomGroupReference('d879d638-e7f1-4a28-a2ab-b4cf2ec7bb4a') } {Id('cb663a55-7c23-431c-b92f-7cd1b2bb1da1')};
    bTimeValid : BOOL { CustomGroupReference('d879d638-e7f1-4a28-a2ab-b4cf2ec7bb4a') } {Id('a833c35b-3ea1-4b2a-b068-2051b4f6b201')};
    nMS : INT { CustomGroupReference('d879d638-e7f1-4a28-a2ab-b4cf2ec7bb4a') } {Id('ea6e97b1-b9ad-49af-a426-0fa38ab26ffc')};
    nHour : INT { CustomGroupReference('d879d638-e7f1-4a28-a2ab-b4cf2ec7bb4a') } {Id('38ed1050-59d1-4396-bf03-b8aea17c9378')};
    nDays : INT { CustomGroupReference('d879d638-e7f1-4a28-a2ab-b4cf2ec7bb4a') } {Id('7805c54d-606c-4a03-92f0-45b2bc4e6a78')};
    TimestampMs : ULINT { CustomGroupReference('d879d638-e7f1-4a28-a2ab-b4cf2ec7bb4a') } {Id('0559e812-68fe-42c6-b1e0-b42bbbfc9d76')};
    i : INT { CustomGroupReference('d879d638-e7f1-4a28-a2ab-b4cf2ec7bb4a') } {Id('7ec15adf-b700-4341-a2c3-f33168454540')};
    nCurrentTimestampMs : ULINT { CustomGroupReference('d879d638-e7f1-4a28-a2ab-b4cf2ec7bb4a') } {Id('85da6c48-e94b-4f0c-a30b-6d1480e7b53e')};
    nLastBlinkMicroseconds : INT { CustomGroupReference('d879d638-e7f1-4a28-a2ab-b4cf2ec7bb4a') } {Id('da205537-b5dc-469b-b99c-e758f52de6df')};
    nCurrentMicroseconds : INT { CustomGroupReference('d879d638-e7f1-4a28-a2ab-b4cf2ec7bb4a') } {Id('d4f0ec62-779b-4dc0-82b5-a89d163c5fd6')};
    PressTimestampMs : BOOL { CustomGroupReference('d879d638-e7f1-4a28-a2ab-b4cf2ec7bb4a') } {Id('a99e92e6-fa03-40ed-bc9f-1fadc5c0c56f')};
    CurrentTimestampMs : BOOL { CustomGroupReference('d879d638-e7f1-4a28-a2ab-b4cf2ec7bb4a') } {Id('cf4bdeb9-944e-4471-9ac8-034bc3ab670a')};
    bTimeParsed : BOOL { CustomGroupReference('d879d638-e7f1-4a28-a2ab-b4cf2ec7bb4a') } {Id('111e3442-1ff1-4dd4-b8af-442cf5c26f34')};
    Valid : BOOL { CustomGroupReference('d879d638-e7f1-4a28-a2ab-b4cf2ec7bb4a') } {Id('8b15ae26-e512-47e1-acb8-c7162f3632a6')};
    INT_TO_ULINT : BOOL { CustomGroupReference('d879d638-e7f1-4a28-a2ab-b4cf2ec7bb4a') } {Id('e497151f-0beb-4bba-bced-536f818e6c6f')};
    Millisecond : INT { CustomGroupReference('d879d638-e7f1-4a28-a2ab-b4cf2ec7bb4a') } {Id('e94126a3-eff3-451f-b81e-3c04fbe87c99')};
    Second : INT { CustomGroupReference('d879d638-e7f1-4a28-a2ab-b4cf2ec7bb4a') } {Id('a7b32ef0-5ea4-4a84-8615-02ae0a0ee8c2')};
    Minute : INT { CustomGroupReference('d879d638-e7f1-4a28-a2ab-b4cf2ec7bb4a') } {Id('96328dad-65c6-46c1-b27a-c16981db8bf8')};
    Hour : INT { CustomGroupReference('d879d638-e7f1-4a28-a2ab-b4cf2ec7bb4a') } {Id('9a24ff45-cc8f-4807-8bbc-7d1a2da63b63')};
    DINT_TO_ULINT : BOOL { CustomGroupReference('d879d638-e7f1-4a28-a2ab-b4cf2ec7bb4a') } {Id('6b7576d9-aed3-4675-9ab5-4376548ff2c5')};
    Days : DINT { CustomGroupReference('d879d638-e7f1-4a28-a2ab-b4cf2ec7bb4a') } {Id('c558866f-8f52-4841-bc1d-6cd71ac139a9')};
    Day : INT { CustomGroupReference('d879d638-e7f1-4a28-a2ab-b4cf2ec7bb4a') } {Id('cee0bbbc-f10b-4dfe-a1af-12b2a55d1cd2')};
    MonthDays11 : DINT { CustomGroupReference('d879d638-e7f1-4a28-a2ab-b4cf2ec7bb4a') } {Id('f8ba89dc-2094-42ce-8a25-aaafc6431308')};
    Month : INT { CustomGroupReference('d879d638-e7f1-4a28-a2ab-b4cf2ec7bb4a') } {Id('51a9e8a8-78a4-4577-910c-81169e3c6f50')};
    MonthDays4 : DINT { CustomGroupReference('d879d638-e7f1-4a28-a2ab-b4cf2ec7bb4a') } {Id('dacea02a-8cdb-46be-b3c8-339ea16fa611')};
    MonthDays2 : DINT { CustomGroupReference('d879d638-e7f1-4a28-a2ab-b4cf2ec7bb4a') } {Id('855d3b6d-0f4c-480a-8f1c-1329942a1461')};
    MonthDays1 : DINT { CustomGroupReference('d879d638-e7f1-4a28-a2ab-b4cf2ec7bb4a') } {Id('e703b079-8c8c-4d0c-9617-25da500a3272')};
    MonthDays6 : DINT { CustomGroupReference('d879d638-e7f1-4a28-a2ab-b4cf2ec7bb4a') } {Id('0120bdca-f7f8-4a56-8c2c-582580363dd0')};
    MonthDays8 : DINT { CustomGroupReference('d879d638-e7f1-4a28-a2ab-b4cf2ec7bb4a') } {Id('58b4f828-5007-4322-bb5d-0f195c4b98a6')};
    MonthDays10 : DINT { CustomGroupReference('d879d638-e7f1-4a28-a2ab-b4cf2ec7bb4a') } {Id('52b07a9c-7b4a-40c2-9e6c-21b97da46201')};
    MonthDays3 : DINT { CustomGroupReference('d879d638-e7f1-4a28-a2ab-b4cf2ec7bb4a') } {Id('5c9cd26b-1638-40cd-beac-0de68a6a6b26')};
    MonthDays5 : DINT { CustomGroupReference('d879d638-e7f1-4a28-a2ab-b4cf2ec7bb4a') } {Id('26e8f3d8-d930-4744-ad4c-47f6d09271f9')};
    MonthDays7 : DINT { CustomGroupReference('d879d638-e7f1-4a28-a2ab-b4cf2ec7bb4a') } {Id('0ea1369b-fad9-42c7-8d18-5742384aacf1')};
    MonthDays9 : DINT { CustomGroupReference('d879d638-e7f1-4a28-a2ab-b4cf2ec7bb4a') } {Id('d90dbc90-d49c-435e-a893-c724f21dda60')};
    Year : INT { CustomGroupReference('d879d638-e7f1-4a28-a2ab-b4cf2ec7bb4a') } {Id('92884857-24e3-4a0f-ba60-e9415c49bb40')};
    MonthDays12 : INT { CustomGroupReference('d879d638-e7f1-4a28-a2ab-b4cf2ec7bb4a') } {Id('84ac20e9-7c2f-47da-93c0-215088391c13')};
    sYear : STRING { CustomGroupReference('d879d638-e7f1-4a28-a2ab-b4cf2ec7bb4a') } {Id('f48f94f1-9b83-4097-96fc-4b719526f9b4')};
    sMonth : STRING { CustomGroupReference('d879d638-e7f1-4a28-a2ab-b4cf2ec7bb4a') } {Id('d62c3366-2ddf-4350-bb4e-f3922cc7b992')};
    sDay : STRING { CustomGroupReference('d879d638-e7f1-4a28-a2ab-b4cf2ec7bb4a') } {Id('e59f804e-d42c-4341-b14b-25cdfef4055a')};
    sHour : STRING { CustomGroupReference('d879d638-e7f1-4a28-a2ab-b4cf2ec7bb4a') } {Id('c6a96e73-a726-40cc-982a-b88a8cb1147d')};
    sMinute : STRING { CustomGroupReference('d879d638-e7f1-4a28-a2ab-b4cf2ec7bb4a') } {Id('17e9b4b6-7a63-44cb-a2ef-e33e2500ad1e')};
    sSecond : STRING { CustomGroupReference('d879d638-e7f1-4a28-a2ab-b4cf2ec7bb4a') } {Id('fa6afaa5-1bed-4ccc-938c-f17052e37b75')};
    nDotPos : INT { CustomGroupReference('d879d638-e7f1-4a28-a2ab-b4cf2ec7bb4a') } {Id('31821420-d110-4ff9-b795-0bce06193bf0')};
    sMS : STRING { CustomGroupReference('d879d638-e7f1-4a28-a2ab-b4cf2ec7bb4a') } {Id('ede553a8-ed38-47b3-9489-2d3e1cb3bad8')};
    nElapsedSincePressMs : ULINT { CustomGroupReference('d879d638-e7f1-4a28-a2ab-b4cf2ec7bb4a') } {Id('ae5f9a75-c2b0-4fe6-ab41-668357300412')};
    bLongPressDetected : BOOL { CustomGroupReference('d879d638-e7f1-4a28-a2ab-b4cf2ec7bb4a') } {Id('42fdab6f-99b5-41c1-a9cf-1c482293dd59')};
    nPressTimestampMs : ULINT { CustomGroupReference('d879d638-e7f1-4a28-a2ab-b4cf2ec7bb4a') } {Id('8c7cc4ba-ed07-4cc9-b2ba-77420aa8000a')};
END_VAR

(* ---- FB1.pou~Code~0000.st ---- *)
BUTTON_VIRTUAL := BUTTON_VIRTUAL AND NOT bLastButtonState;

// регает нажатие
IF (BUTTON_01 OR BUTTON_VIRTUAL) AND NOT bLastButtonState AND TIMER >= 300 AND TIMER <= 5000 THEN
    bIsBlinking := NOT bIsBlinking;
    visual_counter := visual_counter + 1;
END_IF;

IF TIMER < 300 THEN
    MESSAGE := FALSE;
ELSE
    MESSAGE := TRUE;
END_IF;

bLastButtonState := BUTTON_01 OR BUTTON_VIRTUAL;

// мигание
IF bIsBlinking THEN

    counter := counter + 1;

    IF counter >= (TIMER / 10) THEN
        LED := NOT LED;

        IF LED THEN
            tap_counter := tap_counter + 1;
        END_IF;

        counter := 0;
    END_IF;

ELSE
    LED := FALSE;
    counter := 0;
END_IF;

BUTTON_VIRTUAL := FALSE;

(* ---- FB1.pou~Code~0001.st ---- *)
BUTTON_VIRTUAL := BUTTON_VIRTUAL AND NOT bLastButtonState;

IF (BUTTON_01 OR BUTTON_VIRTUAL) AND NOT bLastButtonState AND TIMER >= 300 AND TIMER <= 5000 THEN
    bIsBlinking := NOT bIsBlinking;
    visual_counter := visual_counter + 1;
END_IF

IF TIMER < 300 THEN    //сообщ с ошибкой
    MESSAGE := FALSE;
ELSE
    MESSAGE := TRUE;
END_IF

bLastButtonState := BUTTON_01 OR BUTTON_VIRTUAL;

IF bIsBlinking THEN
    counter := counter + 1;
    TIMER := TIMER / 10;
    IF counter >= TIMER THEN
        LED := NOT LED;
        IF LED = TRUE THEN
            tap_counter := tap_counter + 1;
         END_IF
        counter := 0;
    END_IF
        TIMER := TIMER * 10;
ELSE
    LED := FALSE;
    counter := 0;
END_IF

BUTTON_VIRTUAL := FALSE;

(* ---- FB1.pou~Variables~0000.var ---- *)
{ CustomGroupDefinition('31edb4d9-a441-4cea-9bde-ca4f26605bb2', '') }

VAR_EXTERNAL
    BUTTON_01 : BOOL { CustomGroupReference('31edb4d9-a441-4cea-9bde-ca4f26605bb2') } {Id('09aebbb0-1189-4ff3-8d2d-3695e20b69ed')};
    BUTTON_VIRTUAL : BOOL { CustomGroupReference('31edb4d9-a441-4cea-9bde-ca4f26605bb2') } {Id('546d12ed-b06e-48b0-9d4a-55e62e8e2a03')};
    TIMER : UINT { CustomGroupReference('31edb4d9-a441-4cea-9bde-ca4f26605bb2') } {Id('0a8c6ebd-7c0d-4469-a92d-1805afebcb24')};
    LED : BOOL { CustomGroupReference('31edb4d9-a441-4cea-9bde-ca4f26605bb2') } {Id('dcbdc499-b3fe-498a-803e-2c05b1dc0cbb')};
    MESSAGE : BOOL { CustomGroupReference('31edb4d9-a441-4cea-9bde-ca4f26605bb2') } {Id('ba9b3110-f150-4e05-8ff6-1ce80ba1dd19')};
    tap_counter : UINT { CustomGroupReference('31edb4d9-a441-4cea-9bde-ca4f26605bb2') } {Id('af59b3a0-e3dd-42ee-81fd-37f5e7812363')};
    counter : UINT { CustomGroupReference('31edb4d9-a441-4cea-9bde-ca4f26605bb2') } {Id('6be55703-5707-4767-a30c-47cb2bedbcbe')};
    visual_counter : UINT { CustomGroupReference('31edb4d9-a441-4cea-9bde-ca4f26605bb2') } {Id('b1efa4c6-c926-45f4-9231-0356f4280e0f')};
    bLastButtonState : BOOL { CustomGroupReference('31edb4d9-a441-4cea-9bde-ca4f26605bb2') } {Id('84b4362d-df9f-4bdd-be78-91d7a14ab0d5')};
    bIsBlinking : BOOL { CustomGroupReference('31edb4d9-a441-4cea-9bde-ca4f26605bb2') } {Id('6c780264-d7f1-4c78-a4a9-19327e5d3764')};
    buttonEdge : BOOL { CustomGroupReference('31edb4d9-a441-4cea-9bde-ca4f26605bb2') } {Id('c96592bf-bfab-44ca-b2b8-f77803951dce')};
END_VAR

(* ---- FB1.pou~Variables~0001.var ---- *)
{ CustomGroupDefinition('eb95ad15-efdf-425f-b1f7-cad914f82e05', '') }

VAR_EXTERNAL
    bIsBlinking : BOOL { CustomGroupReference('eb95ad15-efdf-425f-b1f7-cad914f82e05') } {Id('fd348598-50ff-48c3-b6dc-bb9d57c59c48')};
    bLastButtonState : BOOL { CustomGroupReference('eb95ad15-efdf-425f-b1f7-cad914f82e05') } {Id('028e38dd-d89a-4075-8c37-e57d5f3f1be6')};
    BUTTON_01 : BOOL { CustomGroupReference('eb95ad15-efdf-425f-b1f7-cad914f82e05') } {Id('97737f1d-f865-4f7f-b069-c2ca4c75a6e2')};
    BUTTON_VIRTUAL : BOOL { CustomGroupReference('eb95ad15-efdf-425f-b1f7-cad914f82e05') } {Id('c96c8079-8b15-42c0-86ba-3a262873b082')};
    counter : UINT { CustomGroupReference('eb95ad15-efdf-425f-b1f7-cad914f82e05') } {Id('fb87ad38-92cb-4aac-a2de-7bfd96d20931')};
    visual_counter : UINT { CustomGroupReference('eb95ad15-efdf-425f-b1f7-cad914f82e05') } {Id('8d82f5c7-9708-4ece-9127-46b204c4313b')};
    TIMER : UINT { CustomGroupReference('eb95ad15-efdf-425f-b1f7-cad914f82e05') } {Id('91c3396f-74a8-40ad-b2c2-3bd5fd9ed3a2')};
    MESSAGE : BOOL { CustomGroupReference('eb95ad15-efdf-425f-b1f7-cad914f82e05') } {Id('eab0f88a-bcc3-4569-b13e-add472a805f2')};
    LED : BOOL { CustomGroupReference('eb95ad15-efdf-425f-b1f7-cad914f82e05') } {Id('1b446ec7-6ecc-4b5d-bee2-145b4a99ecf5')};
    tap_counter : UINT { CustomGroupReference('eb95ad15-efdf-425f-b1f7-cad914f82e05') } {Id('63809bfb-97a4-4f93-b79b-b0c3badf1e28')};
END_VAR

(* ---- FB2.pou~Code~0000.st ---- *)
TON_Button(IN := BUTTON_01 OR BUTTON_VIRTUAL, PT := T#5S);

IF (BUTTON_01 OR BUTTON_VIRTUAL) AND NOT bLastButtonState AND TIMER >= 300 THEN
    bIsBlinking := NOT bIsBlinking;
    visual_counter := visual_counter + 1;
END_IF

MESSAGE := (TIMER >= 300);

bLastButtonState := BUTTON_01 OR BUTTON_VIRTUAL;

// моргание
IF bIsBlinking THEN
    TON_Blink(IN := TRUE, PT := T#1000MS);
    IF TON_Blink.Q THEN
        LED := NOT LED;
        IF LED THEN
            tap_counter := tap_counter + 1;
        END_IF
        TON_Blink(IN := FALSE); // сброс таймера
    END_IF
ELSE
    LED := FALSE;
    TON_Blink(IN := FALSE);
END_IF

/*
FB22(
    BUTTON_01 := BUTTON_01,

    BUTTON_VIRTUAL := BUTTON_VIRTUAL,
    LED => LED,
    MESSAGE => MESSAGE,
    visual_counter => visual_counter,
    blinkPeriod => HMI_blinkPeriod,
    tap_counter => tap_counter
    );
*/

(* ---- FB2.pou~Code~0001.st ---- *)
TON_Blink(IN := bIsBlinking, PT := T#500ms);

BUTTON_VIRTUAL := BUTTON_VIRTUAL AND NOT bLastButtonState;

IF (BUTTON_01 OR BUTTON_VIRTUAL) AND NOT bLastButtonState AND TIMER >= 300 AND TIMER <= 5000 THEN
    bIsBlinking := NOT bIsBlinking;
    visual_counter := visual_counter + 1;
END_IF

IF TIMER < 300 THEN
    MESSAGE := FALSE;
ELSE
    MESSAGE := TRUE;
END_IF

bLastButtonState := BUTTON_01 OR BUTTON_VIRTUAL;

IF bIsBlinking THEN
    IF TON_Blink.Q THEN
        LED := NOT LED;
        IF LED = TRUE THEN
            tap_counter := tap_counter + 1;
        END_IF
        TON_Blink(IN := FALSE);
        TON_Blink(IN := TRUE);
    END_IF
ELSE
    LED := FALSE;
    TON_Blink(IN := FALSE);
END_IF

BUTTON_VIRTUAL := FALSE;

(* ---- FB2.pou~Variables~0000.var ---- *)
{ CustomGroupDefinition('b4ee16d5-6a89-4b2f-9dbc-11c1b006edaa', '') }

VAR_INPUT
    BUTTON_01 : BOOL { CustomGroupReference('b4ee16d5-6a89-4b2f-9dbc-11c1b006edaa') } {Id('e8cb44b1-14fc-445d-b585-6572cadc6339')};
    BUTTON_VIRTUAL : BOOL { CustomGroupReference('b4ee16d5-6a89-4b2f-9dbc-11c1b006edaa') } {Id('388eae7d-9ad1-4efd-a24e-612b248896d7')};
END_VAR

VAR_OUTPUT
    LED : BOOL { CustomGroupReference('b4ee16d5-6a89-4b2f-9dbc-11c1b006edaa') } {Id('9bd01ebe-8f0f-4e6e-9056-b12d970e4fd3')};
    MESSAGE : BOOL { CustomGroupReference('b4ee16d5-6a89-4b2f-9dbc-11c1b006edaa') } {Id('8fe6c3f6-f2b8-420d-802a-5e31cf30075d')};
    visual_counter : UINT { CustomGroupReference('b4ee16d5-6a89-4b2f-9dbc-11c1b006edaa') } {Id('84a56341-d8bf-48b4-b690-f641237304cb')};
    tap_counter : UINT { CustomGroupReference('b4ee16d5-6a89-4b2f-9dbc-11c1b006edaa') } {Id('3383d3d9-1443-45b3-8b6d-19f8e13be4af')};
END_VAR

VAR
    bLastButtonState : BOOL { CustomGroupReference('b4ee16d5-6a89-4b2f-9dbc-11c1b006edaa') } {Id('a4cbba39-bf2b-4fa4-928c-916492eef580')};
    bIsBlinking : BOOL { CustomGroupReference('b4ee16d5-6a89-4b2f-9dbc-11c1b006edaa') } {Id('6c1af5c5-e500-4b1a-9ada-44c7728415d6')};
    counter : UINT { CustomGroupReference('b4ee16d5-6a89-4b2f-9dbc-11c1b006edaa') } {Id('f7420e70-7723-422f-978c-6ac68a318c26')};
    TON_Button : TON { CustomGroupReference('b4ee16d5-6a89-4b2f-9dbc-11c1b006edaa') } {Id('067fbeae-ecc4-4369-a374-ae7aa32bf966')};
END_VAR

VAR PUBLIC
    TON_Blink : TON { CustomGroupReference('b4ee16d5-6a89-4b2f-9dbc-11c1b006edaa') } {Id('c9fe0adb-dd9d-40bd-9eda-6131e734701b')};
END_VAR

VAR_EXTERNAL
    TIMER : UINT { CustomGroupReference('b4ee16d5-6a89-4b2f-9dbc-11c1b006edaa') } {Id('18525b79-0705-42ff-a041-425de0718181')};
    TIME_TO_DINT : BOOL { CustomGroupReference('b4ee16d5-6a89-4b2f-9dbc-11c1b006edaa') } {Id('d489808e-de79-4910-b332-a53596208153')};
END_VAR

VAR_OUTPUT
    blinkPeriod : UINT { CustomGroupReference('b4ee16d5-6a89-4b2f-9dbc-11c1b006edaa') } {Id('167eec8b-910e-46af-96dc-b3ff765038bc')};
END_VAR

VAR_EXTERNAL
    UINT_TO_TIME : BOOL { CustomGroupReference('b4ee16d5-6a89-4b2f-9dbc-11c1b006edaa') } {Id('50b19a25-87b5-4a40-b95c-e9d877216690')};
    HMI_blinkPeriod : UINT { CustomGroupReference('b4ee16d5-6a89-4b2f-9dbc-11c1b006edaa') } {Id('2a660bd8-b1c4-43e8-83f1-2e75e552f98e')};
END_VAR

(* ---- FUNCTION.pou~Code~0000.st ---- *)
FUNCTI F_ButtonHandler : BOOL
VAR_INPUT
    BUTTON_01      : BOOL;
    BUTTON_VIRTUAL : BOOL;
    TIMER_IN       : INT;
END_VAR
VAR_OUTPUT
    bIsBlinking    : BOOL;
    LED            : BOOL;
    MESSAGE        : BOOL;
    visual_counter : INT;
    tap_counter    : INT;
    TIMER_OUT      : INT;
END_VAR
VAR
    bLastButtonState : BOOL;
    counter          : INT;
    btn_virt         : BOOL;
END_VAR

(* Тело функции *)
btn_virt := BUTTON_VIRTUAL;
btn_virt := btn_virt AND NOT bLastButtonState;

IF (BUTTON_01 OR btn_virt) AND NOT bLastButtonState AND TIMER_IN >= 300 AND TIMER_IN <= 5000 THEN
    bIsBlinking := NOT bIsBlinking;
    visual_counter := visual_counter + 1;
    F_ButtonHandler := TRUE;
ELSE
    F_ButtonHandler := FALSE;
END_IF

IF TIMER_IN < 300 THEN
    MESSAGE := FALSE;
ELSE
    MESSAGE := TRUE;
END_IF

bLastButtonState := BUTTON_01 OR btn_virt;

IF bIsBlinking THEN
    counter := counter + 1;
    TIMER_OUT := TIMER_IN / 10;
    IF counter >= TIMER_OUT THEN
        LED := NOT LED;
        IF LED = TRUE THEN
            tap_counter := tap_counter + 1;
        END_IF
        counter := 0;
    END_IF
    TIMER_OUT := TIMER_OUT * 10;
ELSE
    LED := FALSE;
    counter := 0;
    TIMER_OUT := TIMER_IN;
END_IF

btn_virt := FALSE;

(* ---- ParseRTC_Time.p~Code~0000.st ---- *)
Valid := TRUE;

// чек минимальной длины
IF LEN(sTime) < 22 THEN
    Valid := FALSE;
    RETURN;
END_IF;

// префикс дт# должен быть
IF LEFT(sTime, 3) <> 'DT#' THEN
    Valid := FALSE;
    RETURN;
END_IF;

sYear   := MID(sTime, 4, 4);
sMonth  := MID(sTime, 2, 9);
sDay    := MID(sTime, 2, 12);
sHour   := MID(sTime, 2, 15);
sMinute := MID(sTime, 2, 18);
sSecond := MID(sTime, 2, 21);

// милисекнуды
nDotPos := FIND(sTime, '.');

IF nDotPos > 0 THEN
    sMS := RIGHT(sTime, LEN(sTime) - nDotPos);
ELSE
    sMS := '0';
END_IF;

// преобразование
Year        := STRING_TO_INT(sYear);
Month       := STRING_TO_INT(sMonth);
Day         := STRING_TO_INT(sDay);
Hour        := STRING_TO_INT(sHour);
Minute      := STRING_TO_INT(sMinute);
Second      := STRING_TO_INT(sSecond);
Millisecond := STRING_TO_INT(sMS);

IF LEN(sMS) = 1 THEN
    Millisecond := Millisecond * 100;
ELSIF LEN(sMS) = 2 THEN
    Millisecond := Millisecond * 10;
END_IF;

// тесты
IF Year < 2000 OR Year > 2100 THEN
    Valid := FALSE;
END_IF;

IF Month < 1 OR Month > 12 THEN
    Valid := FALSE;
END_IF;

IF Day < 1 OR Day > 31 THEN
    Valid := FALSE;
END_IF;

IF Hour > 23 THEN
    Valid := FALSE;
END_IF;

IF Minute > 59 THEN
    Valid := FALSE;
END_IF;

IF Second > 59 THEN
    Valid := FALSE;
END_IF;

(* ---- ParseRTC_T~Variables~0000.var ---- *)
{ CustomGroupDefinition('ff027208-816e-4bae-8d60-82950bdd26b4', '') }

VAR_INPUT
    sTime : STRING { CustomGroupReference('ff027208-816e-4bae-8d60-82950bdd26b4') } {Id('370810b9-d8ce-4693-b016-e1c349ea9af9')};
END_VAR

VAR_OUTPUT
    Year : INT { CustomGroupReference('ff027208-816e-4bae-8d60-82950bdd26b4') } {Id('f2a85ef9-6b1d-4cdb-a26a-4599f89fb160')};
    Month : INT { CustomGroupReference('ff027208-816e-4bae-8d60-82950bdd26b4') } {Id('f750a97c-63d8-4e98-8e34-ff9d5a3f442c')};
    Day : INT { CustomGroupReference('ff027208-816e-4bae-8d60-82950bdd26b4') } {Id('815169e4-50f7-4471-82c4-1a268c26556d')};
    Hour : INT { CustomGroupReference('ff027208-816e-4bae-8d60-82950bdd26b4') } {Id('e9aa74bd-29ec-4a14-805a-ce6ad08d0fe5')};
    Minute : INT { CustomGroupReference('ff027208-816e-4bae-8d60-82950bdd26b4') } {Id('39d76eb6-83ee-4ee9-bfc4-ec3771239c59')};
    Second : INT { CustomGroupReference('ff027208-816e-4bae-8d60-82950bdd26b4') } {Id('8002beec-24f4-4f3c-bc58-2549044a082c')};
    Millisecond : INT { CustomGroupReference('ff027208-816e-4bae-8d60-82950bdd26b4') } {Id('bef2f322-384e-477c-9147-44353bd0fd5b')};
    Valid : BOOL { CustomGroupReference('ff027208-816e-4bae-8d60-82950bdd26b4') } {Id('17c29cb7-d74e-4c23-bbc9-132ea5c7f9c0')};
END_VAR

VAR
    sYear : STRING { CustomGroupReference('ff027208-816e-4bae-8d60-82950bdd26b4') } {Id('e4f9359d-58dd-4b80-84e6-714bf6d56bc6')};
    sMonth : STRING { CustomGroupReference('ff027208-816e-4bae-8d60-82950bdd26b4') } {Id('392083cd-2485-4a68-9ac3-12a84e1ab5f9')};
    sDay : STRING { CustomGroupReference('ff027208-816e-4bae-8d60-82950bdd26b4') } {Id('13daf258-6c16-42c0-8010-b1d773bc36a7')};
    sMinute : STRING { CustomGroupReference('ff027208-816e-4bae-8d60-82950bdd26b4') } {Id('513b5860-c258-4629-8897-662158c5bf67')};
    sSecond : STRING { CustomGroupReference('ff027208-816e-4bae-8d60-82950bdd26b4') } {Id('7b1949aa-e429-438b-8367-18dc388d68a0')};
    sHour : STRING { CustomGroupReference('ff027208-816e-4bae-8d60-82950bdd26b4') } {Id('516230af-e994-4c1b-a9c9-f6c72b0d7727')};
    STRING_TO_INT : BOOL { CustomGroupReference('ff027208-816e-4bae-8d60-82950bdd26b4') } {Id('eea7d005-8153-408b-a852-7b34234430b5')};
    sMS : STRING { CustomGroupReference('ff027208-816e-4bae-8d60-82950bdd26b4') } {Id('2e6383b0-294b-474a-8285-344cab278476')};
    nDotPos : INT { CustomGroupReference('ff027208-816e-4bae-8d60-82950bdd26b4') } {Id('fa8b7165-f5c4-4b84-998d-354a66c66966')};
    nLen : INT { CustomGroupReference('ff027208-816e-4bae-8d60-82950bdd26b4') } {Id('2639a40c-b33c-461e-b5a5-7ba6dedb91ad')};
    nMinute : INT { CustomGroupReference('ff027208-816e-4bae-8d60-82950bdd26b4') } {Id('86abf6a8-7959-4f76-97ea-ead3797c9cdc')};
    nHour : INT { CustomGroupReference('ff027208-816e-4bae-8d60-82950bdd26b4') } {Id('48cca547-1d1f-4e92-8a3b-e408207d64d1')};
    nDay : INT { CustomGroupReference('ff027208-816e-4bae-8d60-82950bdd26b4') } {Id('a2868c9d-fb26-4cc5-b5b9-739609f44cf7')};
    nMonth : INT { CustomGroupReference('ff027208-816e-4bae-8d60-82950bdd26b4') } {Id('46d375c6-1e58-4462-8a32-09ca3d14506a')};
    nYear : INT { CustomGroupReference('ff027208-816e-4bae-8d60-82950bdd26b4') } {Id('7e93e88b-a364-46ff-b433-8f078dd5a72c')};
    nSecond : INT { CustomGroupReference('ff027208-816e-4bae-8d60-82950bdd26b4') } {Id('1f4e089c-d02f-40d4-984d-f8d875afc53e')};
    nMS : INT { CustomGroupReference('ff027208-816e-4bae-8d60-82950bdd26b4') } {Id('4e3827c9-a372-4274-a293-f12a4c0f2486')};
END_VAR

VAR_EXTERNAL
    TRIM : BOOL { CustomGroupReference('ff027208-816e-4bae-8d60-82950bdd26b4') } {Id('7e8fd91a-6666-4f1c-b8eb-3a0792942019')};
END_VAR

(* ---- s.pou~Variables~0000.var ---- *)
{ CustomGroupDefinition('fb84caa8-36a3-47d9-8bf0-95ff0e8a7b24', '') }

VAR_INPUT
    sTime : INT { CustomGroupReference('fb84caa8-36a3-47d9-8bf0-95ff0e8a7b24') } {Id('acdbddae-a692-4e5d-9dbe-b74ee2dc18a1')};
END_VAR

VAR
    Year : INT { CustomGroupReference('fb84caa8-36a3-47d9-8bf0-95ff0e8a7b24') } {Id('82cdfda3-5439-4fe5-8269-74290bfe88f4')};
    Month : INT { CustomGroupReference('fb84caa8-36a3-47d9-8bf0-95ff0e8a7b24') } {Id('906dff29-8c6c-4597-93a7-ce7fe5950296')};
    Day : INT { CustomGroupReference('fb84caa8-36a3-47d9-8bf0-95ff0e8a7b24') } {Id('e8eac52d-d3ce-4d33-9b87-b8758997dbb2')};
    Hour : INT { CustomGroupReference('fb84caa8-36a3-47d9-8bf0-95ff0e8a7b24') } {Id('1edf8d32-8150-4a96-9b46-5199747f10d5')};
    Minute : INT { CustomGroupReference('fb84caa8-36a3-47d9-8bf0-95ff0e8a7b24') } {Id('ba519d36-5300-41de-872b-f3f7f1efe725')};
    Second : INT { CustomGroupReference('fb84caa8-36a3-47d9-8bf0-95ff0e8a7b24') } {Id('551380c9-3eb3-4b47-b945-c24b93d28d98')};
    Millisecond : INT { CustomGroupReference('fb84caa8-36a3-47d9-8bf0-95ff0e8a7b24') } {Id('107b29f2-c4a5-4110-9037-362a1a5b792b')};
    Valid : BOOL { CustomGroupReference('fb84caa8-36a3-47d9-8bf0-95ff0e8a7b24') } {Id('8e80c4a1-4908-4947-81ae-8cf582c29b7b')};
END_VAR

(* ---- TimeStamp.pou~Code~0000.st ---- *)
MonthDays1 := 31;
MonthDays2 := 28;
MonthDays3 := 31;
MonthDays4 := 30;
MonthDays5 := 31;
MonthDays6 := 30;
MonthDays7 := 31;
MonthDays8 := 31;
MonthDays9 := 30;
MonthDays10 := 31;
MonthDays11 := 30;
MonthDays12 := 31;

IF ((Year MOD 4 = 0) AND (Year MOD 100 <> 0)) OR (Year MOD 400 = 0) THEN
    MonthDays2 := 29;
END_IF;

Days := Days + 123;

FOR i := 1970 TO Year - 1 DO
    IF ((i MOD 4 = 0) AND (i MOD 100 <> 0)) OR (i MOD 400 = 0) THEN
        Days := Days + 366;
    ELSE
        Days := Days + 365;
    END_IF;
END_FOR;

IF Month > 1 THEN Days := Days + MonthDays1; END_IF;
IF Month > 2 THEN Days := Days + MonthDays2; END_IF;
IF Month > 3 THEN Days := Days + MonthDays3; END_IF;
IF Month > 4 THEN Days := Days + MonthDays4; END_IF;
IF Month > 5 THEN Days := Days + MonthDays5; END_IF;
IF Month > 6 THEN Days := Days + MonthDays6; END_IF;
IF Month > 7 THEN Days := Days + MonthDays7; END_IF;
IF Month > 8 THEN Days := Days + MonthDays8; END_IF;
IF Month > 9 THEN Days := Days + MonthDays9; END_IF;
IF Month > 10 THEN Days := Days + MonthDays10; END_IF;
IF Month > 11 THEN Days := Days + MonthDays11; END_IF;

Days := Days + (Day - 1);

// Сдвиг на 123 дня

TimestampMs :=
    DINT_TO_ULINT(Days) * 86400000 +
    INT_TO_ULINT(Hour) * 3600000 +
    INT_TO_ULINT(Minute) * 60000 +
    INT_TO_ULINT(Second) * 1000 +
    INT_TO_ULINT(Millisecond);

(* ---- TimeStamp.~Variables~0000.var ---- *)
{ CustomGroupDefinition('86cfc347-5607-405e-9afb-cdf64c624017', '') }

VAR_INPUT
    Year : INT { CustomGroupReference('86cfc347-5607-405e-9afb-cdf64c624017') } {Id('70bb0202-eabc-4b23-b47f-a6f7e5414afd')};
    Month : INT { CustomGroupReference('86cfc347-5607-405e-9afb-cdf64c624017') } {Id('1526e0f8-9578-48d4-a9d6-29e3b3618252')};
    Day : INT { CustomGroupReference('86cfc347-5607-405e-9afb-cdf64c624017') } {Id('ec238d01-6f01-4b66-ab25-b704ff77bb9e')};
    Hour : INT { CustomGroupReference('86cfc347-5607-405e-9afb-cdf64c624017') } {Id('3bf774c5-a55c-47bd-9c26-29b2707f6ef6')};
    Minute : INT { CustomGroupReference('86cfc347-5607-405e-9afb-cdf64c624017') } {Id('073ce2b5-4e3d-41bc-9abe-a6c9f777258c')};
    Second : INT { CustomGroupReference('86cfc347-5607-405e-9afb-cdf64c624017') } {Id('275fd2ff-8ce6-4c4e-bbeb-fe12829f83b8')};
    Millisecond : INT { CustomGroupReference('86cfc347-5607-405e-9afb-cdf64c624017') } {Id('d06b8f1b-9532-4a1a-8bb4-6c535709f9b6')};
END_VAR

VAR_OUTPUT
    TimestampMs : ULINT { CustomGroupReference('86cfc347-5607-405e-9afb-cdf64c624017') } {Id('5e18ebce-5e26-4b86-9e7f-f8ec5f1422bd')};
END_VAR

VAR
    Days : DINT { CustomGroupReference('86cfc347-5607-405e-9afb-cdf64c624017') } {Id('524b0be8-9baa-42cc-a1e2-966c2e57d860')};
    i : INT { CustomGroupReference('86cfc347-5607-405e-9afb-cdf64c624017') } {Id('fe576651-cf45-4d2c-8bff-d4df8445a046')};
    MonthDays1 : INT { CustomGroupReference('86cfc347-5607-405e-9afb-cdf64c624017') } {Id('5118764f-25aa-4ff2-8234-e1f57d2d3e7f')};
    MonthDays2 : INT { CustomGroupReference('86cfc347-5607-405e-9afb-cdf64c624017') } {Id('1ab2c56b-4c75-491f-bc29-ba333d315062')};
    MonthDays3 : INT { CustomGroupReference('86cfc347-5607-405e-9afb-cdf64c624017') } {Id('da0ae2d6-ed19-4086-82f5-b40a8f12c65e')};
    MonthDays4 : INT { CustomGroupReference('86cfc347-5607-405e-9afb-cdf64c624017') } {Id('f7d125cf-0ee3-4eec-ba26-263707c2f6a0')};
    MonthDays5 : INT { CustomGroupReference('86cfc347-5607-405e-9afb-cdf64c624017') } {Id('b603cf9d-1f56-4a42-b4c1-3b09e89ea432')};
    MonthDays6 : INT { CustomGroupReference('86cfc347-5607-405e-9afb-cdf64c624017') } {Id('771bdd4c-dc7b-4c62-b652-ef435ad0e955')};
    MonthDays7 : INT { CustomGroupReference('86cfc347-5607-405e-9afb-cdf64c624017') } {Id('1845af22-1825-4e78-ac82-ea807130fa88')};
    MonthDays8 : INT { CustomGroupReference('86cfc347-5607-405e-9afb-cdf64c624017') } {Id('de581b35-b327-4c73-a2a3-747ffbcb89e2')};
    MonthDays9 : INT { CustomGroupReference('86cfc347-5607-405e-9afb-cdf64c624017') } {Id('bbd68693-4310-4cd0-a465-0ae910676efb')};
    MonthDays10 : INT { CustomGroupReference('86cfc347-5607-405e-9afb-cdf64c624017') } {Id('31269d78-8529-40db-ab50-81e3ba7a4a27')};
    MonthDays11 : INT { CustomGroupReference('86cfc347-5607-405e-9afb-cdf64c624017') } {Id('f6bb2d1f-c419-40c8-aa57-aa863895640a')};
    MonthDays12 : INT { CustomGroupReference('86cfc347-5607-405e-9afb-cdf64c624017') } {Id('33197ee2-7fcb-4191-9aab-a3195d4db147')};
END_VAR

VAR_EXTERNAL
    TIME_TO_DINT : BOOL { CustomGroupReference('86cfc347-5607-405e-9afb-cdf64c624017') } {Id('fd94956a-b23a-4bb5-b728-0efea7ad6a04')};
END_VAR

(* ---- UTC_in_Second.p~Code~0000.st ---- *)
// ---------------------------------------------------------------------
// Тело функционального блока
// ---------------------------------------------------------------------

// 1. Получение времени

IF UseManualRTC THEN
    sTime := ManualRTC;
    bRTC_Ready := TRUE;
ELSE
    fbRTC(EN := TRUE, CDT => sTime, Q => bRTC_Ready);
END_IF;

// 2. Парсинг строки времени

bTimeValid := TRUE;

IF LEN(sTime) < 22 THEN
    bTimeValid := FALSE;
ELSE
    IF LEFT(sTime, 3) <> 'DT#' THEN
        bTimeValid := FALSE;
    ELSE
        sYear   := MID(sTime, 4, 4);
        sMonth  := MID(sTime, 2, 9);
        sDay    := MID(sTime, 2, 12);
        sHour   := MID(sTime, 2, 15);
        sMinute := MID(sTime, 2, 18);
        sSecond := MID(sTime, 2, 21);

        nDotPos := FIND(sTime, '.');

        IF nDotPos > 0 THEN
            sMS := RIGHT(sTime, LEN(sTime) - nDotPos);
        ELSE
            sMS := '0';
        END_IF;

        nYear   := STRING_TO_INT(sYear);
        nMonth  := STRING_TO_INT(sMonth);
        nDay    := STRING_TO_INT(sDay);
        nHour   := STRING_TO_INT(sHour);
        nMinute := STRING_TO_INT(sMinute);
        nSecond := STRING_TO_INT(sSecond);
        nMS     := STRING_TO_INT(sMS);

        IF LEN(sMS) = 1 THEN
            nMS := nMS * 100;
        ELSIF LEN(sMS) = 2 THEN
            nMS := nMS * 10;
        END_IF;

        IF nYear < 2000 OR nYear > 2100 THEN bTimeValid := FALSE; END_IF;
        IF nMonth < 1 OR nMonth > 12 THEN bTimeValid := FALSE; END_IF;
        IF nDay < 1 OR nDay > 31 THEN bTimeValid := FALSE; END_IF;
        IF nHour > 23 THEN bTimeValid := FALSE; END_IF;
        IF nMinute > 59 THEN bTimeValid := FALSE; END_IF;
        IF nSecond > 59 THEN bTimeValid := FALSE; END_IF;
    END_IF;
END_IF;

// 3. Расчет дней от 1970

nDays := 0;

FOR i := 1970 TO nYear - 1 DO
    IF ((i MOD 4 = 0) AND (i MOD 100 <> 0)) OR (i MOD 400 = 0) THEN
        nDays := nDays + 366;
    ELSE
        nDays := nDays + 365;
    END_IF;
END_FOR;

IF ((nYear MOD 4 = 0) AND (nYear MOD 100 <> 0)) OR (nYear MOD 400 = 0) THEN
    nMonthDays2 := 29;
ELSE
    nMonthDays2 := 28;
END_IF;

IF nMonth > 1 THEN nDays := nDays + nMonthDays1; END_IF;
IF nMonth > 2 THEN nDays := nDays + nMonthDays2; END_IF;
IF nMonth > 3 THEN nDays := nDays + nMonthDays3; END_IF;
IF nMonth > 4 THEN nDays := nDays + nMonthDays4; END_IF;
IF nMonth > 5 THEN nDays := nDays + nMonthDays5; END_IF;
IF nMonth > 6 THEN nDays := nDays + nMonthDays6; END_IF;
IF nMonth > 7 THEN nDays := nDays + nMonthDays7; END_IF;
IF nMonth > 8 THEN nDays := nDays + nMonthDays8; END_IF;
IF nMonth > 9 THEN nDays := nDays + nMonthDays9; END_IF;
IF nMonth > 10 THEN nDays := nDays + nMonthDays10; END_IF;
IF nMonth > 11 THEN nDays := nDays + nMonthDays11; END_IF;

nDays := nDays + (nDay - 1);

// 4. Перевод в миллисекунды

IF bTimeValid THEN

    TimestampMs :=
        DINT_TO_ULINT(nDays) * 86400000 +
        INT_TO_ULINT(nHour) * 3600000 +
        INT_TO_ULINT(nMinute) * 60000 +
        INT_TO_ULINT(nSecond) * 1000 +
        INT_TO_ULINT(nMS);

    // Часовой пояс (в часах)
IF TimezoneOffset > 0 THEN
    TimestampMs := TimestampMs + INT_TO_ULINT(TimezoneOffset) * 3600000;
ELSIF TimezoneOffset < 0 THEN
    TimestampMs := TimestampMs - INT_TO_ULINT(ABS(TimezoneOffset)) * 3600000;
END_IF;

    Valid := TRUE;

ELSE

    TimestampMs := 0;
    Valid := FALSE;

END_IF;

// 5. Обработка мигания

IF BlinkReset THEN
    bIsBlinking := FALSE;
    visual_counter := 0;
    tap_counter := 0;
    LED := FALSE;
    nLastBlink := 0;
    bWaitForRelease := FALSE;
END_IF;

(* ---- UTC_in_Sec~Variables~0000.var ---- *)
{ CustomGroupDefinition('3b278276-b7cf-49df-9310-d7f9b6ebd036', '') }

VAR_INPUT
    LEN : BOOL { CustomGroupReference('3b278276-b7cf-49df-9310-d7f9b6ebd036') } {Id('8d6770c3-4fa7-4591-8913-e22d7308c1f9')};
END_VAR

VAR_EXTERNAL
    sTime : STRING { CustomGroupReference('3b278276-b7cf-49df-9310-d7f9b6ebd036') } {Id('57e24803-524f-4a34-ba8a-b77423891213')};
END_VAR

VAR_OUTPUT
    Valid : BOOL { CustomGroupReference('3b278276-b7cf-49df-9310-d7f9b6ebd036') } {Id('2c0b8204-1976-4346-bf68-4f004ddc3b58')};
    TimestampMs : ULINT { CustomGroupReference('3b278276-b7cf-49df-9310-d7f9b6ebd036') } {Id('70cc4bd4-80af-4401-8cac-9d1c71a5fe44')};
END_VAR

VAR
    sYear : STRING { CustomGroupReference('3b278276-b7cf-49df-9310-d7f9b6ebd036') } {Id('931b130c-ca28-4a28-ae57-109b438232aa')};
    sMonth : STRING { CustomGroupReference('3b278276-b7cf-49df-9310-d7f9b6ebd036') } {Id('07c60b4e-348a-4af1-8cf5-dd6ea12d0b3e')};
    sHour : STRING { CustomGroupReference('3b278276-b7cf-49df-9310-d7f9b6ebd036') } {Id('ea345062-e35d-4c03-9edf-2a0ddbc5e2c4')};
    sDay : STRING { CustomGroupReference('3b278276-b7cf-49df-9310-d7f9b6ebd036') } {Id('80eb27d9-3ebd-440d-99aa-59ffc489b769')};
    sMinute : STRING { CustomGroupReference('3b278276-b7cf-49df-9310-d7f9b6ebd036') } {Id('5dbd2db2-9d44-4c9a-8644-cc3f59393a31')};
    sSecond : STRING { CustomGroupReference('3b278276-b7cf-49df-9310-d7f9b6ebd036') } {Id('b8d96fe8-0a41-4952-874f-7e4ce94ffc04')};
    nDotPos : INT { CustomGroupReference('3b278276-b7cf-49df-9310-d7f9b6ebd036') } {Id('43aab87a-42f6-497b-ab35-2a636348fbc3')};
    sMS : STRING { CustomGroupReference('3b278276-b7cf-49df-9310-d7f9b6ebd036') } {Id('fd2b1ba0-3c87-4dee-ab85-ba21a6a446aa')};
    Year : INT { CustomGroupReference('3b278276-b7cf-49df-9310-d7f9b6ebd036') } {Id('e2360734-ab99-455c-93e8-5e4c47d87b31')};
    Month : INT { CustomGroupReference('3b278276-b7cf-49df-9310-d7f9b6ebd036') } {Id('9965d299-4b6e-4164-bb30-ad7a40f8a335')};
    Hour : INT { CustomGroupReference('3b278276-b7cf-49df-9310-d7f9b6ebd036') } {Id('5878f747-eae7-4528-b61a-6e4dce7b0cb7')};
    Minute : INT { CustomGroupReference('3b278276-b7cf-49df-9310-d7f9b6ebd036') } {Id('1bce9a80-89f7-4d19-b2ee-07c333b60940')};
    Day : INT { CustomGroupReference('3b278276-b7cf-49df-9310-d7f9b6ebd036') } {Id('7d6db6a5-977b-4e8a-9a0c-b49b754886de')};
    Second : INT { CustomGroupReference('3b278276-b7cf-49df-9310-d7f9b6ebd036') } {Id('ff1c5c23-717d-4ace-bfc1-b974571af825')};
    Millisecond : INT { CustomGroupReference('3b278276-b7cf-49df-9310-d7f9b6ebd036') } {Id('6f9a1f9c-ff25-4d8a-b145-8fa1cacc147a')};
    MonthDays1 : INT { CustomGroupReference('3b278276-b7cf-49df-9310-d7f9b6ebd036') } {Id('8ea123db-38f2-4013-ac7d-cb021428cbaf')};
    MonthDays5 : INT { CustomGroupReference('3b278276-b7cf-49df-9310-d7f9b6ebd036') } {Id('469196d8-51ef-4cbc-9da5-dd06cd9758b4')};
    MonthDays8 : INT { CustomGroupReference('3b278276-b7cf-49df-9310-d7f9b6ebd036') } {Id('c41e239d-a006-4798-b976-fd8e05a7e948')};
    MonthDays6 : INT { CustomGroupReference('3b278276-b7cf-49df-9310-d7f9b6ebd036') } {Id('b3dc4ea3-90c8-4311-81e8-c63be88d5ad3')};
    MonthDays9 : INT { CustomGroupReference('3b278276-b7cf-49df-9310-d7f9b6ebd036') } {Id('4796c50b-444e-453a-8df3-6724a99983a2')};
    MonthDays12 : INT { CustomGroupReference('3b278276-b7cf-49df-9310-d7f9b6ebd036') } {Id('4e7a6a5f-f80a-4f65-a4b3-905fdbc18814')};
    MonthDays10 : INT { CustomGroupReference('3b278276-b7cf-49df-9310-d7f9b6ebd036') } {Id('d0a249ff-7353-4c2d-8422-6c070ff260fa')};
    MonthDays7 : INT { CustomGroupReference('3b278276-b7cf-49df-9310-d7f9b6ebd036') } {Id('1ee760d2-5b67-432f-94e2-724b3a776a39')};
    MonthDays4 : INT { CustomGroupReference('3b278276-b7cf-49df-9310-d7f9b6ebd036') } {Id('341beb9b-c740-4251-b6d6-303bd10b04ed')};
    MonthDays2 : INT { CustomGroupReference('3b278276-b7cf-49df-9310-d7f9b6ebd036') } {Id('06742f12-859d-4dc2-b961-2439cc7c6423')};
    MonthDays11 : INT { CustomGroupReference('3b278276-b7cf-49df-9310-d7f9b6ebd036') } {Id('56b7d9e0-9cde-419c-ab91-a6ab0f6d3957')};
    MonthDays3 : INT { CustomGroupReference('3b278276-b7cf-49df-9310-d7f9b6ebd036') } {Id('f42d9edd-06ae-4c62-862e-32e410afac61')};
    Days : INT { CustomGroupReference('3b278276-b7cf-49df-9310-d7f9b6ebd036') } {Id('8c7f8e10-e5a3-4161-a103-0fdd1c57bdd0')};
    i : INT { CustomGroupReference('3b278276-b7cf-49df-9310-d7f9b6ebd036') } {Id('f30fc678-7fa9-486e-968f-cee05a925eb8')};
    fbRTC : RTC_S { CustomGroupReference('3b278276-b7cf-49df-9310-d7f9b6ebd036') } {Id('b843552d-1d57-4733-b2ec-b62f5d05bbb7')};
    sYearTemp : STRING { CustomGroupReference('3b278276-b7cf-49df-9310-d7f9b6ebd036') } {Id('5fbb706c-8ea7-400d-961f-a25751e16c27')};
    sMonthTemp : STRING { CustomGroupReference('3b278276-b7cf-49df-9310-d7f9b6ebd036') } {Id('6e787a00-8ae1-42e3-97ef-6b0dcfd97f66')};
    sDayTemp : STRING { CustomGroupReference('3b278276-b7cf-49df-9310-d7f9b6ebd036') } {Id('6f0c9eda-f8c3-49dd-8c0d-f7890696ff14')};
    sHourTemp : STRING { CustomGroupReference('3b278276-b7cf-49df-9310-d7f9b6ebd036') } {Id('ec57f270-2e70-4497-9302-ff4fd6d882ee')};
    sMinuteTemp : STRING { CustomGroupReference('3b278276-b7cf-49df-9310-d7f9b6ebd036') } {Id('1939b24a-be25-4c91-b00a-12db0851901e')};
END_VAR

VAR_INPUT
    EN_RTC : BOOL { CustomGroupReference('3b278276-b7cf-49df-9310-d7f9b6ebd036') } {Id('69162fa0-7492-4adf-8ddf-2789fba5e529')};
END_VAR

VAR_EXTERNAL
    bRTC_Ready : BOOL { CustomGroupReference('3b278276-b7cf-49df-9310-d7f9b6ebd036') } {Id('36439ad9-84a0-48aa-aa24-04e40e870101')};
END_VAR

VAR
    sINT_TO_STRING : BOOL { CustomGroupReference('3b278276-b7cf-49df-9310-d7f9b6ebd036') } {Id('0190df65-ddc6-4623-af82-b9e0ef8027c5')};
    sSecondTemp : BOOL { CustomGroupReference('3b278276-b7cf-49df-9310-d7f9b6ebd036') } {Id('77806555-c500-43c3-8122-272a80464a90')};
    MonthDays : BOOL { CustomGroupReference('3b278276-b7cf-49df-9310-d7f9b6ebd036') } {Id('40e51b3c-85fb-4e34-a42c-1ebc170e5864')};
    MS : INT { CustomGroupReference('3b278276-b7cf-49df-9310-d7f9b6ebd036') } {Id('e4546e1e-835f-44c5-80c8-2943a1a20ceb')};
    nYear : INT { CustomGroupReference('3b278276-b7cf-49df-9310-d7f9b6ebd036') } {Id('3b2d767c-fabe-4096-887e-b47e217c11a7')};
    nDays : INT { CustomGroupReference('3b278276-b7cf-49df-9310-d7f9b6ebd036') } {Id('adf0cd1a-f830-4055-a297-6969ef91d2f8')};
    nMonth : INT { CustomGroupReference('3b278276-b7cf-49df-9310-d7f9b6ebd036') } {Id('e79f0a96-7bdd-4c09-be00-fee7ecfa6731')};
    nDay : INT { CustomGroupReference('3b278276-b7cf-49df-9310-d7f9b6ebd036') } {Id('f31da16d-9a8e-4156-8224-16da0a3d35b2')};
    fbParseTime : ParseRTC_Time { CustomGroupReference('3b278276-b7cf-49df-9310-d7f9b6ebd036') } {Id('105578e8-8941-437f-9b3f-3c834f413ab2')};
    nHour : INT { CustomGroupReference('3b278276-b7cf-49df-9310-d7f9b6ebd036') } {Id('d2117bf4-5837-48e5-910e-84629f333295')};
    nMinute : INT { CustomGroupReference('3b278276-b7cf-49df-9310-d7f9b6ebd036') } {Id('439d5659-28fe-476a-872c-e6810d761671')};
    nSecond : INT { CustomGroupReference('3b278276-b7cf-49df-9310-d7f9b6ebd036') } {Id('80220a70-d710-46db-91b1-199a6d566a6e')};
    nMS : INT { CustomGroupReference('3b278276-b7cf-49df-9310-d7f9b6ebd036') } {Id('84196a6e-6e86-4dba-abed-184b9d9f3d92')};
    bTimeValid : BOOL { CustomGroupReference('3b278276-b7cf-49df-9310-d7f9b6ebd036') } {Id('e9fb3372-2492-42a4-876e-1e48886a869f')};
    nMonthDays1 : INT { CustomGroupReference('3b278276-b7cf-49df-9310-d7f9b6ebd036') } {Id('5d05df01-dd6e-4c59-8e36-83954c44d2fd')};
    nMonthDays2 : INT { CustomGroupReference('3b278276-b7cf-49df-9310-d7f9b6ebd036') } {Id('345a8cc5-e23b-4ff7-8029-1650f573b20b')};
    nMonthDays4 : INT { CustomGroupReference('3b278276-b7cf-49df-9310-d7f9b6ebd036') } {Id('46202a87-db8e-4a5f-9150-fecaf7b5716f')};
    nMonthDays7 : INT { CustomGroupReference('3b278276-b7cf-49df-9310-d7f9b6ebd036') } {Id('c9e3ea73-3602-4914-998a-52c14ce4345b')};
    nMonthDays9 : INT { CustomGroupReference('3b278276-b7cf-49df-9310-d7f9b6ebd036') } {Id('2d576936-c5a1-4a61-bb70-bda9d3659500')};
    nMonthDays8 : INT { CustomGroupReference('3b278276-b7cf-49df-9310-d7f9b6ebd036') } {Id('9b2ab0a3-5263-4eab-b5ad-62e0797279d2')};
    nMonthDays10 : INT { CustomGroupReference('3b278276-b7cf-49df-9310-d7f9b6ebd036') } {Id('a1e25079-646b-4880-9359-54979dcfbb36')};
    nMonthDays11 : INT { CustomGroupReference('3b278276-b7cf-49df-9310-d7f9b6ebd036') } {Id('e2011caa-7db9-4c00-ac5c-e1ca39ec0584')};
    nMonthDays3 : INT { CustomGroupReference('3b278276-b7cf-49df-9310-d7f9b6ebd036') } {Id('fc4a0175-d7b5-4aaf-a7ae-505b74999737')};
    nMonthDays5 : INT { CustomGroupReference('3b278276-b7cf-49df-9310-d7f9b6ebd036') } {Id('1ae5419f-81a8-480b-aca2-3ab04dd5bf8e')};
    nMonthDays6 : INT { CustomGroupReference('3b278276-b7cf-49df-9310-d7f9b6ebd036') } {Id('b97973c8-7c52-4b7e-8df0-5870a960cbc1')};
END_VAR

VAR_OUTPUT
    bIsBlinking : BOOL { CustomGroupReference('3b278276-b7cf-49df-9310-d7f9b6ebd036') } {Id('3c332540-4c4f-4e81-b1dc-d18d2a37acfb')};
    LED : BOOL { CustomGroupReference('3b278276-b7cf-49df-9310-d7f9b6ebd036') } {Id('4e3602ef-2168-4547-9054-a7dea89d41e8')};
END_VAR

VAR
    bWaitForRelease : BOOL { CustomGroupReference('3b278276-b7cf-49df-9310-d7f9b6ebd036') } {Id('a68a3c25-3fb3-4182-a201-01ed43e53017')};
    nLastBlink : INT { CustomGroupReference('3b278276-b7cf-49df-9310-d7f9b6ebd036') } {Id('8a06fba6-f022-4b76-9ddf-f263e13af148')};
    tap_counter : INT { CustomGroupReference('3b278276-b7cf-49df-9310-d7f9b6ebd036') } {Id('eb76768e-7803-48ef-9e81-34239926b21f')};
    visual_counter : INT { CustomGroupReference('3b278276-b7cf-49df-9310-d7f9b6ebd036') } {Id('9c940fbc-ca3e-4e80-aec3-d69c29707bbb')};
END_VAR

VAR_INPUT
    BlinkReset : BOOL { CustomGroupReference('3b278276-b7cf-49df-9310-d7f9b6ebd036') } {Id('f780c3eb-aefa-4d80-b7ef-7fbabba8cb70')};
END_VAR

VAR_EXTERNAL
    TimeZone : INT { CustomGroupReference('3b278276-b7cf-49df-9310-d7f9b6ebd036') } {Id('fd8e153f-31c3-441b-990c-0e5b0fa48b58')};
    nTimeZoneOffset : INT { CustomGroupReference('3b278276-b7cf-49df-9310-d7f9b6ebd036') } {Id('533862a9-0891-4cbf-811a-6dbc86b91b2e')};
END_VAR

VAR
    bConvertToMS : BOOL { CustomGroupReference('3b278276-b7cf-49df-9310-d7f9b6ebd036') } {Id('ae3fb4e7-bf10-4790-bd99-6cdd422ddf27')};
END_VAR

VAR_EXTERNAL
    sCustomDate : STRING { CustomGroupReference('3b278276-b7cf-49df-9310-d7f9b6ebd036') } {Id('eedff408-d8cc-446f-b322-f971dccfa6c6')};
END_VAR

VAR
    nPos : INT { CustomGroupReference('3b278276-b7cf-49df-9310-d7f9b6ebd036') } {Id('efcd1563-5640-4f22-90ed-3c6cbb08c48c')};
    sHh : STRING { CustomGroupReference('3b278276-b7cf-49df-9310-d7f9b6ebd036') } {Id('7462822a-d8dd-4686-9b09-4d71416d8e18')};
    sYyyy : STRING { CustomGroupReference('3b278276-b7cf-49df-9310-d7f9b6ebd036') } {Id('4b03d1fe-b6db-49fb-8a32-b96d2eef122a')};
    nCustomMonth : INT { CustomGroupReference('3b278276-b7cf-49df-9310-d7f9b6ebd036') } {Id('d4ce5159-1035-4fb3-bca5-8cb294b5bd2b')};
    nCustomDays : INT { CustomGroupReference('3b278276-b7cf-49df-9310-d7f9b6ebd036') } {Id('d9e74d6e-ce2a-40d1-8155-264c0525e572')};
    nCustomYear : INT { CustomGroupReference('3b278276-b7cf-49df-9310-d7f9b6ebd036') } {Id('8fa7cff9-3035-475b-a546-ab0b148e808a')};
    nCustomSecond : INT { CustomGroupReference('3b278276-b7cf-49df-9310-d7f9b6ebd036') } {Id('b66ac111-94e9-43c5-8da9-c2627fcaf34e')};
    nCustomMinute : INT { CustomGroupReference('3b278276-b7cf-49df-9310-d7f9b6ebd036') } {Id('3baa8834-2414-437f-8b6f-f5c1f2bdf57e')};
    nCustomHour : INT { CustomGroupReference('3b278276-b7cf-49df-9310-d7f9b6ebd036') } {Id('88fc4d65-7e14-40c2-91eb-3064f2a0115b')};
    nCustomDay : INT { CustomGroupReference('3b278276-b7cf-49df-9310-d7f9b6ebd036') } {Id('23822389-cc9d-4dd9-bad7-d0c660422744')};
    sSTRING_TO_INT : BOOL { CustomGroupReference('3b278276-b7cf-49df-9310-d7f9b6ebd036') } {Id('25ab36db-77ab-4f00-96e9-adeae8c696fd')};
    sMm : STRING { CustomGroupReference('3b278276-b7cf-49df-9310-d7f9b6ebd036') } {Id('29fded2d-bd39-46b0-a944-915747c1b563')};
    sSs : STRING { CustomGroupReference('3b278276-b7cf-49df-9310-d7f9b6ebd036') } {Id('535696f1-7817-4c36-b2ad-3f2984840ca6')};
    sDd : STRING { CustomGroupReference('3b278276-b7cf-49df-9310-d7f9b6ebd036') } {Id('85ee92cd-42b8-4496-9809-0ac30835a7b4')};
    sMn : STRING { CustomGroupReference('3b278276-b7cf-49df-9310-d7f9b6ebd036') } {Id('6abcf799-6876-4860-b222-10780c45846e')};
    nTempMS : ULINT { CustomGroupReference('3b278276-b7cf-49df-9310-d7f9b6ebd036') } {Id('9d07504c-a27b-4150-91a2-75cf4509b8fc')};
END_VAR

VAR_EXTERNAL
    ulInputMS : ULINT { CustomGroupReference('3b278276-b7cf-49df-9310-d7f9b6ebd036') } {Id('d9505d5a-a8b0-43e9-9cf7-226d1d39ea66')};
    sOutputDate : STRING { CustomGroupReference('3b278276-b7cf-49df-9310-d7f9b6ebd036') } {Id('e7c5913a-3710-4d0b-934b-e2dbcda7cd2f')};
END_VAR

VAR
    sTemp : STRING { CustomGroupReference('3b278276-b7cf-49df-9310-d7f9b6ebd036') } {Id('9e6ae635-445a-4bbf-a005-9dfdc4f41652')};
    sDINT_TO_STRING : BOOL { CustomGroupReference('3b278276-b7cf-49df-9310-d7f9b6ebd036') } {Id('9a9d356f-54ad-4897-b6db-3ccc187010ba')};
    DaysInMonth AT %I* : INT { CustomGroupReference('3b278276-b7cf-49df-9310-d7f9b6ebd036') } {Id('4d13c785-6bc4-44b1-80e0-43a1c407399e')};
END_VAR

VAR_EXTERNAL
    sTmp : BOOL { CustomGroupReference('3b278276-b7cf-49df-9310-d7f9b6ebd036') } {Id('33783de1-11ee-4c10-8389-e955f41a1a85')};
    sTmp2 : BOOL { CustomGroupReference('3b278276-b7cf-49df-9310-d7f9b6ebd036') } {Id('f6323b1c-ad59-46f9-8149-bb8c38f49731')};
    sYy : STRING { CustomGroupReference('3b278276-b7cf-49df-9310-d7f9b6ebd036') } {Id('f4be37f2-b054-452f-bbd5-f26a591e82ae')};
    sMo : STRING { CustomGroupReference('3b278276-b7cf-49df-9310-d7f9b6ebd036') } {Id('130c9d8c-1b43-419e-8b85-366a53d4f490')};
    nMonthDays : INT { CustomGroupReference('3b278276-b7cf-49df-9310-d7f9b6ebd036') } {Id('824b2f22-0277-4584-ad9d-8cd81b71739f')};
    UseManualRTC : BOOL { CustomGroupReference('3b278276-b7cf-49df-9310-d7f9b6ebd036'), TRANSLATE } {Id('e6de7347-2ad9-43ca-898e-901e0bd61e7d')};
    ManualRTC : STRING { CustomGroupReference('3b278276-b7cf-49df-9310-d7f9b6ebd036') } {Id('fe49dd22-b5bd-4596-b05a-d6324f5aa3c4')};
    TimezoneOffset : INT { CustomGroupReference('3b278276-b7cf-49df-9310-d7f9b6ebd036') } {Id('f9d0c43b-ede4-4914-b959-ea8d39dad0e1')};
END_VAR
